# B&R Automation Studio project RTFProj (part 2)

#### calculation_displacementOfAxes.c
```c
/*********************************************************************************************
* B&R Automation - Perfection in Automation (https://www.br-automation.com)
    ******************************************************************************************
    * Program 	    : Master's Thesis - Soccer Table (Simulation)
    * Author  	    : Roman Parak
    * Created 	    : date ...
	* University    : Brno University of Technology(BUT)
	* Faculty       : Faculty of Mechanical Engineering(FME)
	* Study Program : Applied Computer Science and Control
	* Institute     : Institute of Automation and Computer Science
**********************************************************************************************
* Implementation OF PROGRAM simulation(rp_library/rp_funcx1/rp_functions.c)
**********************************************************************************************/

/************************************* LIBRARIES *********************************************/
#include <bur/plctypes.h>
#include <math.h>
#include <string.h>

#ifdef __cplusplus
	extern "C"
	{
#endif
	#include "rp_funcx1.h"
#ifdef __cplusplus
	};
#endif

void calculation_displacementOfAxes(struct calculation_displacementOfAxes* c_dOA)
{
	REAL max_dispOfD[4], min_dispOfD[4], max_posOfD[4], min_posOfD[4], matrix_posOfCPU[4][5], real_disp[4];
	REAL velocity[4], acceleration[4], deceleration[4];
	REAL aux_velocity[4], aux_acceleration[4];
	REAL aux_time;
	UDINT auxiliary_str;
	USINT i_rC, i_rCn, i, j, i_out, i_chRD, i_chRDn, i_chRDnn;

	struct calculation_realCrossing calc_rC;
	struct choosing_rightDummy ch_rightD;

	// Ceilings of the axes
	// Axes
	max_posOfD[0] = 820;
	max_posOfD[1] = 3050;
	max_posOfD[2] = 3050;
	max_posOfD[3] = 3055;

	min_posOfD[0] = -950;
	min_posOfD[1] = -3050;
	min_posOfD[2] = -3050;
	min_posOfD[3] = -3055;
	// Dummies
	max_dispOfD[0] = 820;
	max_dispOfD[1] = 1850;
	max_dispOfD[2] = 650;
	max_dispOfD[3] = 955;

	min_dispOfD[0] = -950;
	min_dispOfD[1] = -1850;
	min_dispOfD[2] = -650;
	min_dispOfD[3] = -955;
	// Actual positions of dummies CPU
	// goalkeeper
	matrix_posOfCPU[0][0] = 0 + c_dOA->act_displacementCPU[0];
	// defender
	matrix_posOfCPU[1][0] = -1200 + c_dOA->act_displacementCPU[1];
	matrix_posOfCPU[1][1] = 1200 + c_dOA->act_displacementCPU[1];
	// midfielder
	matrix_posOfCPU[2][0] = -2400 + c_dOA->act_displacementCPU[2];
	matrix_posOfCPU[2][1] = -1200 + c_dOA->act_displacementCPU[2];
	matrix_posOfCPU[2][2] = 0 + c_dOA->act_displacementCPU[2];
	matrix_posOfCPU[2][3] = 1200 + c_dOA->act_displacementCPU[2];
	matrix_posOfCPU[2][4] = 2400 + c_dOA->act_displacementCPU[2];
	// forward
	matrix_posOfCPU[3][0] = -2100 + c_dOA->act_displacementCPU[3];
	matrix_posOfCPU[3][1] = 0 + c_dOA->act_displacementCPU[3];
	matrix_posOfCPU[3][2] = 2100 + c_dOA->act_displacementCPU[3];

	// function block -> output is a array of real crossing
	calc_rC.tilted = c_dOA->tilted;
	auxiliary_str = (UDINT) strcpy(calc_rC.specific_direction,c_dOA->specific_direction);
	for(i_rC = 0; i_rC < (int)(sizeof(max_posOfD)/sizeof(max_posOfD[0])); i_rC++){
		calc_rC.act_posOfAxesCPU_Y[i_rC]		 = c_dOA->act_posOfAxesCPU_Y[i_rC];
		calc_rC.act_posOfAxesHUM_Y[i_rC]		 = c_dOA->act_posOfAxesHUM_Y[i_rC];
		calc_rC.count_axesIntersectionHUM[i_rC]  = c_dOA->count_axesIntersectionHUM[i_rC];
		calc_rC.reversed_HUM[i_rC]				 = c_dOA->reversed_HUM[i_rC];
	}
	for(i_rCn = 0; i_rCn < (int)(sizeof(c_dOA->act_posOfDummiesH)/sizeof(c_dOA->act_posOfDummiesH[0])); i_rCn++){
		calc_rC.act_posOfDummiesH[i_rCn] = c_dOA->act_posOfDummiesH[i_rCn];
	}
	calc_rC.x_posOfBall[0] = c_dOA->x_posOfBall[0];
	calc_rC.x_posOfBall[1] = c_dOA->x_posOfBall[1];
	calculation_realCrossing(&calc_rC);

	for(i = 0; i < (int)(sizeof(calc_rC.real_cross)/sizeof(calc_rC.real_cross[0])); i++){
		if(calc_rC.real_cross[i] > max_posOfD[i]){
			real_disp[i] = max_dispOfD[i];
		}else if(calc_rC.real_cross[i] < min_posOfD[i]){
			real_disp[i] = min_dispOfD[i];
		}else {
			ch_rightD.index      = i;
			ch_rightD.real_cross = calc_rC.real_cross[i];

			for(i_chRD = 0; i_chRD < (int)(sizeof(max_dispOfD)/sizeof(max_dispOfD[0])); i_chRD++){
				ch_rightD.max_dispOfD[i_chRD] = max_dispOfD[i_chRD];
				ch_rightD.min_dispOfD[i_chRD] = min_dispOfD[i_chRD];
			}

			for(i_chRDn = 0; i_chRDn < (int)(sizeof(max_dispOfD)/sizeof(max_dispOfD[0])); i_chRDn++){
				for(i_chRDnn = 0; i_chRDnn <= (int)(sizeof(max_dispOfD)/sizeof(max_dispOfD[0]));i_chRDnn++){
					ch_rightD.matrix_posOfCPU[i_chRDn][i_chRDnn] = matrix_posOfCPU[i_chRDn][i_chRDnn];
				}
			}
			choosing_rightDummy(&ch_rightD);

			real_disp[i] = ch_rightD.actual_displacement;
		}
	}// end for{i}

	for(i_out = 0; i_out < (int)(sizeof(calc_rC.real_cross)/sizeof(calc_rC.real_cross[0])); i_out++){
		// max velocity = 29000, max acceleration = 489 000
		aux_time = 0.07;
		aux_velocity[i_out] = fabs(fabs(real_disp[i_out]) - fabs(c_dOA->act_displacementCPU[i_out]))/c_dOA->time_axisIntersection[i_out];

		if(aux_velocity[i_out] > 29000){
			velocity[i_out] 		= fabs(fabs(real_disp[i_out]) - fabs(c_dOA->act_displacementCPU[i_out]))/aux_time;
			aux_acceleration[i_out] = velocity[i_out]/c_dOA->time_axisIntersection[i_out];

			if(aux_acceleration[i_out] > 489000){
				acceleration[i_out] = 489000;
				deceleration[i_out] = 489000;
			}else{
				acceleration[i_out] = aux_acceleration[i_out];
				deceleration[i_out] = aux_acceleration[i_out];
			}
		}else{
			velocity[i_out] 		= aux_velocity[i_out];
			aux_acceleration[i_out] = velocity[i_out]/c_dOA->time_axisIntersection[i_out];

			if(aux_acceleration[i_out] > 489000){
				acceleration[i_out] = 489000;
				deceleration[i_out] = 489000;
			}else{
				acceleration[i_out] = aux_acceleration[i_out];
				deceleration[i_out] = aux_acceleration[i_out];
			}
		}

		c_dOA->displacement[i_out] = real_disp[i_out];
		c_dOA->velocity[i_out] 	   = velocity[i_out];
		c_dOA->acceleration[i_out] = acceleration[i_out];
		c_dOA->deceleration[i_out] = deceleration[i_out];
	}// end for{i_out}

}// end function

void calculation_realCrossing(struct calculation_realCrossing* c_rC)
{
	REAL matrix_posOfHUM[4][5], matrix_crossH_Iter[0][5], matrix_crossH_Pos[0][5];
	REAL predicted_pos;
	USINT number_ofD[4], count_crossH, count_calcH;
	USINT iteration, iteration_positionH;
	USINT j, j_null, i_yC, i_yCn, i_cNC, i_out, r;
	BOOL auxiliary_bool,auxiliary_boolNo2;
	UDINT auxiliary_str;

	struct calculation_newCrossing calc_newC;

	auxiliary_bool 	  = 0;
	auxiliary_boolNo2 = 0;
	// Actual positions of dummies HUMAN
	// goalkeeper
	matrix_posOfHUM[0][0] = c_rC->act_posOfDummiesH[0];
	// defender
	matrix_posOfHUM[1][0] = c_rC->act_posOfDummiesH[1];
	matrix_posOfHUM[1][1] = c_rC->act_posOfDummiesH[2];
	// midfielder
	matrix_posOfHUM[2][0] = c_rC->act_posOfDummiesH[3];
	matrix_posOfHUM[2][1] = c_rC->act_posOfDummiesH[4];
	matrix_posOfHUM[2][2] = c_rC->act_posOfDummiesH[5];
	matrix_posOfHUM[2][3] = c_rC->act_posOfDummiesH[6];
	matrix_posOfHUM[2][4] = c_rC->act_posOfDummiesH[7];
	// forward
	matrix_posOfHUM[3][0] = c_rC->act_posOfDummiesH[8];
	matrix_posOfHUM[3][1] = c_rC->act_posOfDummiesH[9];
	matrix_posOfHUM[3][2] = c_rC->act_posOfDummiesH[10];

	number_ofD[0] = 1;
	number_ofD[1] = 2;
	number_ofD[2] = 5;
	number_ofD[3] = 3;

	calc_newC.reversed_HUM = 1;

	count_crossH   = c_rC->count_axesIntersectionHUM[0];
	count_calcH    = 5 - count_crossH;

	if(count_calcH == 0){
		iteration = 1;
	}else{
		iteration = count_calcH;
	}

	if(count_calcH < 5){
		for(j = 0; j < number_ofD[count_calcH - 1]; j++){
			if(c_rC->reversed_HUM[count_calcH - 1] == 0){
				if(((matrix_posOfHUM[count_calcH - 1][j] <= c_rC->act_posOfAxesHUM_Y[count_calcH - 1] + 100) && (matrix_posOfHUM[count_calcH - 1][j] >= c_rC->act_posOfAxesHUM_Y[count_calcH - 1])) && (matrix_posOfHUM[count_calcH - 1][j] != c_rC->act_posOfAxesHUM_Y[count_calcH - 1])){
					matrix_crossH_Iter[0][j] = count_calcH;
					matrix_crossH_Pos[0][j]  = fabs(fabs(matrix_posOfHUM[count_calcH - 1][j]) - fabs(c_rC->act_posOfAxesHUM_Y[count_calcH - 1]));
				}else if(((matrix_posOfHUM[count_calcH - 1][j] >= c_rC->act_posOfAxesHUM_Y[count_calcH - 1] - 100) && (matrix_posOfHUM[count_calcH - 1][j] <= c_rC->act_posOfAxesHUM_Y[count_calcH - 1])) && (matrix_posOfHUM[count_calcH - 1][j] != c_rC->act_posOfAxesHUM_Y[count_calcH - 1])){
					matrix_crossH_Iter[0][j] = count_calcH;
					matrix_crossH_Pos[0][j]  = (-1)*fabs(fabs(matrix_posOfHUM[count_calcH - 1][j]) - fabs(c_rC->act_posOfAxesHUM_Y[count_calcH - 1]));
				}else if(matrix_posOfHUM[count_calcH - 1][j] == c_rC->act_posOfAxesHUM_Y[count_calcH - 1]){
					matrix_crossH_Iter[0][j] = count_calcH;
					matrix_crossH_Pos[0][j]  = 0;
				}else{
					matrix_crossH_Iter[0][j] = 0;
					matrix_crossH_Pos[0][j]  = 0;
				}
			}else{
				matrix_crossH_Iter[0][j] = 0;
				matrix_crossH_Pos[0][j]  = 0;
			}
		}

		for(r = 0; r < number_ofD[count_calcH - 1]; r++){
			if(matrix_crossH_Iter[0][r] != 0){
				calc_newC.reversed_HUM = 0;
			}
		}
		for(j_null = 0; j_null < number_ofD[count_calcH - 1]; j_null++){
			if(matrix_crossH_Iter[0][j_null] != 0){
				auxiliary_bool 		= 1;
				predicted_pos  		= matrix_crossH_Pos[0][j_null];
				iteration_positionH = matrix_crossH_Iter[0][j_null];
			}
		}

		if(auxiliary_bool == 0){
			if(c_rC->tilted == 0){
				predicted_pos 		= 0;
				iteration_positionH = iteration;
			}else{
				auxiliary_boolNo2 = 1;
				for(i_yCn = 0; i_yCn < (int)(sizeof(c_rC->act_posOfAxesCPU_Y)/sizeof(c_rC->act_posOfAxesCPU_Y[0])); i_yCn++){
					c_rC->real_cross[i_yCn] = c_rC->act_posOfAxesCPU_Y[i_yCn];
				}
			}
		}

	}else{
		if(c_rC->tilted == 0){
			calc_newC.reversed_HUM = 0;
			predicted_pos 		   = 0;
			iteration_positionH    = count_calcH;
		}else{
			auxiliary_boolNo2 = 1;
			for(i_yC = 0; i_yC < (int)(sizeof(c_rC->act_posOfAxesCPU_Y)/sizeof(c_rC->act_posOfAxesCPU_Y[0])); i_yC++){
				c_rC->real_cross[i_yC] = c_rC->act_posOfAxesCPU_Y[i_yC];
			}
		}
	}// end : if(count_calcH < 5)

	if(auxiliary_boolNo2 != 1){
		auxiliary_str = (UDINT) strcpy(calc_newC.specific_direction,c_rC->specific_direction);
		calc_newC.iteration 		 = iteration_positionH;
		calc_newC.predicted_position = predicted_pos;
		for(i_cNC = 0; i_cNC < (int)(sizeof(c_rC->act_posOfAxesCPU_Y)/sizeof(c_rC->act_posOfAxesCPU_Y[0])); i_cNC++){
			calc_newC.act_posOfAxesCPU_Y[i_cNC] = c_rC->act_posOfAxesCPU_Y[i_cNC];
			calc_newC.act_posOfAxesHUM_Y[i_cNC] = c_rC->act_posOfAxesHUM_Y[i_cNC];
		}
		calc_newC.x_posOfBall[0] = c_rC->x_posOfBall[0];
		calc_newC.x_posOfBall[1] = c_rC->x_posOfBall[1];
		calculation_newCrossing(&calc_newC);

		for(i_out = 0; i_out < (int)(sizeof(c_rC->act_posOfAxesCPU_Y)/sizeof(c_rC->act_posOfAxesCPU_Y[0])); i_out++){
			c_rC->real_cross[i_out] = calc_newC.new_cross[i_out];
		}
	}// end if(auxiliary_boolNo2 != 1)
}// end function

void calculation_newCrossing(struct calculation_newCrossing* c_nC)
{
	INT gk_max, gk_min, value;
	SINT iteration;
	DINT resultUP, resultLF, resultDOWN, resultRH;
	REAL y_crossGK, y_crossDF, y_crossMD, y_crossFW;

	// initial max goalkeeper
	gk_max = 820;
	gk_min = -950;

	resultUP   = strcmp(c_nC->specific_direction, "up_backward");
	resultLF   = strcmp(c_nC->specific_direction, "left");
	resultDOWN = strcmp(c_nC->specific_direction, "down_backward");
	resultRH   = strcmp(c_nC->specific_direction, "right");

	if(resultUP == 0 || resultLF == 0){
		value = 200;
	}else if(resultDOWN == 0 || resultRH == 0){
		value = -200;
	}else{
		value = 200;
	}

	if(c_nC->iteration > 4){
		iteration = 4;
	}else{
		iteration = c_nC->iteration;
	}

	switch(iteration){
		case 1:
			{
				y_crossFW = c_nC->act_posOfAxesCPU_Y[4];
				y_crossMD = y_crossFW + value;
				y_crossDF = y_crossMD + value;
				y_crossGK = y_crossDF + value;

				if(fabs(y_crossGK) > fabs(y_crossFW)){
					y_crossGK = y_crossFW - value;
				}

				if(fabs(y_crossMD) < fabs(y_crossFW)){
					y_crossMD = y_crossFW - value;
					y_crossDF = y_crossMD - value;
				}
			}
			break;
		case 2:
			{
				if(c_nC->x_posOfBall[0] >= 9800){
					y_crossFW = c_nC->act_posOfAxesHUM_Y[iteration] - c_nC->predicted_position;
					y_crossMD = y_crossFW + value;
					y_crossDF = y_crossMD + value;
					y_crossGK = y_crossDF + value;

					if(fabs(y_crossGK) > fabs(y_crossFW)){
						y_crossGK = y_crossFW - value;
					}

					if(fabs(y_crossMD) < fabs(y_crossFW)){
						y_crossMD = y_crossFW - value;
						y_crossDF = y_crossMD - value;
					}
				}else{
					y_crossFW = c_nC->act_posOfAxesHUM_Y[3] - c_nC->predicted_position;
					y_crossMD = y_crossFW + value;
					y_crossDF = y_crossMD + value;
					y_crossGK = y_crossDF + value;

					if(fabs(y_crossGK) > fabs(y_crossFW)){
						y_crossGK = y_crossFW - value;
					}

					if(fabs(y_crossMD) < fabs(y_crossFW)){
						y_crossMD = y_crossFW - value;
						y_crossDF = y_crossMD - value;
					}
				}
			}
			break;
		case 3:
			{
				if(c_nC->reversed_HUM == 1){
					y_crossFW = c_nC->act_posOfAxesHUM_Y[3] - c_nC->predicted_position;
					y_crossMD = y_crossFW + value;
				}else{
					y_crossFW = c_nC->act_posOfAxesHUM_Y[3] - c_nC->predicted_position;
					y_crossMD = y_crossFW + value;
				}

				y_crossDF = y_crossMD + value;
				y_crossGK = y_crossFW + value;

				if(fabs(y_crossGK) > fabs(y_crossFW)){
					y_crossGK = y_crossFW - value;
				}

				if(fabs(y_crossMD) < fabs(y_crossFW)){
					y_crossMD = y_crossFW - value;
					y_crossDF = y_crossMD - value;
				}
			}
			break;
		case 4:
			{
				if(c_nC->x_posOfBall[0] >= 5300){
					if(c_nC->reversed_HUM == 1){
						y_crossFW = c_nC->act_posOfAxesCPU_Y[3] - c_nC->predicted_position;
						y_crossMD = c_nC->act_posOfAxesCPU_Y[2] - c_nC->predicted_position;
						y_crossDF = y_crossMD + value;
						y_crossGK = y_crossFW + value;
					}else{
						y_crossFW = c_nC->act_posOfAxesCPU_Y[3] - c_nC->predicted_position;
						y_crossMD = c_nC->act_posOfAxesCPU_Y[2] - c_nC->predicted_position;
						y_crossDF = y_crossMD - c_nC->predicted_position;
						y_crossGK = y_crossFW + value;

					}

					if(fabs(y_crossGK) > fabs(y_crossFW)){
						y_crossGK = y_crossFW - value;
					}
					if(fabs(y_crossMD) < fabs(y_crossFW)){
						y_crossDF = y_crossMD - value;
					}
				}else{
					y_crossFW = c_nC->act_posOfAxesCPU_Y[3] - c_nC->predicted_position;
					y_crossMD = c_nC->act_posOfAxesCPU_Y[2] - c_nC->predicted_position;
					y_crossDF = y_crossMD - c_nC->predicted_position;
					y_crossGK = y_crossFW + value;
				}

				if(c_nC->x_posOfBall[0] <= 2300){
					y_crossGK = c_nC->act_posOfAxesCPU_Y[0];
				}
			}
			break;
	}// end switch

	if(y_crossGK > gk_max){
		y_crossGK = y_crossDF - 200;
	}else if(y_crossGK < gk_min){
		y_crossGK = y_crossDF + 200;
	}

	c_nC->new_cross[0] = y_crossGK;
	c_nC->new_cross[1] = y_crossDF;
	c_nC->new_cross[2] = y_crossMD;
	c_nC->new_cross[3] = y_crossFW;

}// end function

void choosing_rightDummy(struct choosing_rightDummy* ch_rD)
{
	REAL real_cross;
	REAL d_DFD[2],d_MDD[5], d_FWD[3];
	USINT i_df, i_md, i_fw;
	struct calculete_min calc_m;

	switch(ch_rD->index){
		case 0:
			{
				real_cross 				   = ch_rD->real_cross;
				ch_rD->actual_displacement = real_cross;
			}
			break;
		case 1:
			{
				d_DFD[0] = fabs((fabs(ch_rD->matrix_posOfCPU[ch_rD->index][0]) + ch_rD->real_cross));
				d_DFD[1] = fabs((ch_rD->matrix_posOfCPU[ch_rD->index][1] - ch_rD->real_cross));

				for(i_df = 0; i_df < (int)(sizeof(calc_m.cmp_num)/sizeof(calc_m.cmp_num[0])); i_df++){
					if(i_df < ((int)(sizeof(d_DFD)/sizeof(d_DFD[0])))){
						calc_m.cmp_num[i_df] = d_DFD[i_df];
					}else{
						calc_m.cmp_num[i_df] = 5000;
					}
				}
			}
			break;
		case 2:
			{
				d_MDD[0] = fabs((fabs(ch_rD->matrix_posOfCPU[ch_rD->index][0]) + ch_rD->real_cross));
				d_MDD[1] = fabs((fabs(ch_rD->matrix_posOfCPU[ch_rD->index][1]) + ch_rD->real_cross));
				d_MDD[2] = fabs((ch_rD->real_cross));
				d_MDD[3] = fabs((fabs(ch_rD->matrix_posOfCPU[ch_rD->index][3]) - ch_rD->real_cross));
				d_MDD[4] = fabs((fabs(ch_rD->matrix_posOfCPU[ch_rD->index][4]) - ch_rD->real_cross));

				for(i_md = 0; i_md < (int)(sizeof(calc_m.cmp_num)/sizeof(calc_m.cmp_num[0])); i_md++){
					calc_m.cmp_num[i_md] = d_MDD[i_md];
				}
			}
			break;
		case 3:
			{
				d_FWD[0] = fabs((fabs(ch_rD->matrix_posOfCPU[ch_rD->index][0]) + ch_rD->real_cross));
				d_FWD[1] = fabs((ch_rD->real_cross));
				d_FWD[2] = fabs((fabs(ch_rD->matrix_posOfCPU[ch_rD->index][2]) - ch_rD->real_cross));

				for(i_fw = 0; i_fw < (int)(sizeof(calc_m.cmp_num)/sizeof(calc_m.cmp_num[0])); i_fw++){
					if(i_fw < ((int)(sizeof(d_FWD)/sizeof(d_FWD[0])))){
						calc_m.cmp_num[i_fw] = d_FWD[i_fw];
					}else{
						calc_m.cmp_num[i_fw] = 5000;
					}
				}
			}
			break;
	}// end switch

	if(ch_rD->index != 0){
		calculete_min(&calc_m);

		if(calc_m.number > ch_rD->max_dispOfD[ch_rD->index]){
			real_cross = ch_rD->max_dispOfD[ch_rD->index];
		}else if(calc_m.number < ch_rD->min_dispOfD[ch_rD->index]){
			real_cross = ch_rD->min_dispOfD[ch_rD->index];
		}else{
			real_cross = calc_m.number;
		}

		if(ch_rD->real_cross > ch_rD->matrix_posOfCPU[ch_rD->index][calc_m.index]){
			ch_rD->actual_displacement = real_cross;
		}else{
			ch_rD->actual_displacement = (-1)*real_cross;
		}
	}
}// end function

void calculete_min(struct calculete_min* c_m)
{
	REAL min;
	USINT i, idx;

	min = 30000;
	for(i = 0; i < (int)(sizeof(c_m->cmp_num)/sizeof(c_m->cmp_num[0])); i++){
		if(c_m->cmp_num[i] < min){
			min = c_m->cmp_num[i];
			idx = i;
		}
	}

	c_m->index  = idx;
	c_m->number = min;
}// end function
```

#### measurement_ofScore.c
```c
#include <bur/plctypes.h>
#include <bur/plc.h>
#include <astime.h>
#include <string.h>
#include <math.h>

#ifdef __cplusplus
	extern "C"
	{
#endif
	#include "rp_funcx1.h"
#ifdef __cplusplus
	};
#endif
void initialization(struct measurement_ofScore* m_oS);

void measurement_ofScore(struct measurement_ofScore* m_oS)
{

    if(!m_oS->start_measurement){
        initialization(m_oS);
    }

    switch(m_oS->Internal.state){
        case 0:
            {
                if(m_oS->Internal.counter <= 0){
                    m_oS->Internal.counter = 0;
                }

                m_oS->Internal.results[0]   = strcmp(m_oS->PLAYER1_NAME, "");
                m_oS->Internal.results[1]   = strcmp(m_oS->PLAYER2_NAME, "");

                if(m_oS->start_measurement == 1 && m_oS->Error == 0){
                    if(m_oS->Internal.results[0] == 0 && m_oS->Internal.results[1] == 0){
                        m_oS->Internal.auxiliary_str[5] = (UDINT) strcpy(m_oS->PLAYER1_NAME,"PLAYER 1");
                        m_oS->Internal.auxiliary_str[6] = (UDINT) strcpy(m_oS->PLAYER2_NAME,"PLAYER 2");
                    }
                    // CPU NAME
                    m_oS->Internal.auxiliary_str[7] = (UDINT) strcpy(m_oS->team_nameCPU,"B&R ROBOT");
                    // HUMAN NAME
                    strcpy(m_oS->Internal.string[5],m_oS->PLAYER1_NAME);
                    strcpy(m_oS->Internal.string[6]," \n \t& \n");
                    strcpy(m_oS->Internal.string[8], m_oS->PLAYER2_NAME);
                    m_oS->Internal.auxiliary_str[8] = (UDINT) strcat(m_oS->Internal.string[5], m_oS->Internal.string[6]);
                    strcpy(m_oS->Internal.string[7], m_oS->Internal.string[5]);
                    m_oS->Internal.auxiliary_str[9] = (UDINT) strcat(m_oS->Internal.string[7], m_oS->Internal.string[8]);
                    m_oS->Internal.auxiliary_str[10] = (UDINT) strcpy(m_oS->team_nameHUM,m_oS->Internal.auxiliary_str[9]);
                    // CHANGE STATE
                    m_oS->Internal.state = 1;
                }else if(m_oS->Error == 1){
                    m_oS->Internal.state = 5;
                }else if(m_oS->pause == 1){
                    m_oS->Internal.before_state = m_oS->Internal.state;
                    m_oS->Internal.state = 6;
                }else{
                    m_oS->Internal.state = 0;
                }
            }
            break;
        case 1:
            {
                if(m_oS->sens_wicket_CPU == 1){
                    m_oS->count_goals_CPU++;
                    m_oS->sens_wicket_CPU = 0;
                }

                if(m_oS->sens_wicket_HUM == 1){
                    m_oS->count_goals_HUM++;
                    m_oS->sens_wicket_HUM = 0;
                }

                if((m_oS->count_goals_HUM - m_oS->count_goals_CPU) == 0){
                    m_oS->probability_CPU = 50;
                    m_oS->probability_HUM = 50;
                }else if((m_oS->count_goals_HUM - m_oS->count_goals_CPU) < 0){
                    if(fabs((m_oS->count_goals_HUM - m_oS->count_goals_CPU)) <= 5){
                        m_oS->probability_CPU = 50 + fabs((m_oS->count_goals_HUM - m_oS->count_goals_CPU))*10;
                        m_oS->probability_HUM = 100 - m_oS->probability_CPU;
                    }else{
                        m_oS->probability_CPU = 100;
                        m_oS->probability_HUM = 0;
                    }
                }else{
                    if(fabs((m_oS->count_goals_HUM - m_oS->count_goals_CPU)) <= 5){
                        m_oS->probability_HUM = 50 + fabs((m_oS->count_goals_HUM - m_oS->count_goals_CPU))*10;
                        m_oS->probability_CPU = 100 - m_oS->probability_HUM;
                    }else{
                        m_oS->probability_HUM = 100;
                        m_oS->probability_CPU = 0;
                    }
                }
                if(((m_oS->count_goals_CPU + m_oS->count_goals_HUM) == 10) && m_oS->Error == 0){
                    m_oS->Internal.state             = 2;
                    m_oS->Internal.write_matchInfo   = 1;
                }else if(m_oS->exit_game == 1 ){
                    m_oS->Internal.state = 3;
                }else if(m_oS->restart_measurement == 1){
                    m_oS->Internal.state = 4;
                }else if(m_oS->Error == 1){
                    m_oS->Internal.state = 5;
                }else if(m_oS->pause == 1){
                    m_oS->Internal.before_state = m_oS->Internal.state;
                    m_oS->Internal.state = 6;
                }else{
                    m_oS->Internal.state = 1;
                }

            }
            break;
        case 2:
            {
                if(m_oS->Internal.write_matchInfo == 1){
                    // call FB : Get time and date
                    m_oS->Internal.UtcDTStructureGetTime_1.enable = 1;
                    m_oS->Internal.UtcDTStructureGetTime_1.pDTStructure = (UDINT) &m_oS->Internal.DTStruct;
                    UtcDTStructureGetTime(&m_oS->Internal.UtcDTStructureGetTime_1);
                    ascDTStructure((UDINT) &m_oS->Internal.DTStruct, (UDINT) &m_oS->Internal.string[0], m_oS->Internal.length);
                    // write time and date into the variable
                    m_oS->Internal.auxiliary_str[0] = (UDINT) strcpy(m_oS->match_informations.date[m_oS->Internal.counter],m_oS->Internal.string[0]);
                    // write score
                    m_oS->match_informations.score_CPU[m_oS->Internal.counter] = m_oS->count_goals_CPU;
                    m_oS->match_informations.score_HUM[m_oS->Internal.counter] = m_oS->count_goals_HUM;
                    // write name of B&R team
                    m_oS->Internal.auxiliary_str[1] = (UDINT) strcpy(m_oS->match_informations.team_name_CPU[m_oS->Internal.counter],"B&R ROBOT");
                    // write names of both players
                    strcpy(m_oS->Internal.string[1],m_oS->PLAYER1_NAME);
                    strcpy(m_oS->Internal.string[2]," & ");
                    strcpy(m_oS->Internal.string[4], m_oS->PLAYER2_NAME);
                    m_oS->Internal.auxiliary_str[2] = (UDINT) strcat(m_oS->Internal.string[1], m_oS->Internal.string[2]);
                    strcpy(m_oS->Internal.string[3], m_oS->Internal.string[1]);
                    m_oS->Internal.auxiliary_str[3] = (UDINT) strcat(m_oS->Internal.string[3], m_oS->Internal.string[4]);
                    m_oS->Internal.auxiliary_str[4] = (UDINT) strcpy(m_oS->match_informations.team_name_HUM[m_oS->Internal.counter],m_oS->Internal.auxiliary_str[3]);

                    m_oS->Internal.counter++;
                    m_oS->Internal.write_matchInfo = 0;
                }

                if(m_oS->exit_game == 1){
                    m_oS->Internal.state = 3;
                }else if(m_oS->restart_measurement == 1){
                    m_oS->Internal.state = 4;
                }else if(m_oS->Error == 1){
                    m_oS->Internal.state = 5;
                }else if(m_oS->pause == 1){
                    m_oS->Internal.before_state = m_oS->Internal.state;
                    m_oS->Internal.state = 6;
                }else{
                    m_oS->Internal.state = 2;
                }
            }
            break;
        case 3:
            {
                // exit game
                m_oS->start_measurement   = 0;
                m_oS->exit_game           = 0;
                m_oS->restart_measurement = 0;
                m_oS->count_goals_CPU     = 0;
                m_oS->count_goals_HUM     = 0;

                m_oS->Internal.e_r_str[0] = (UDINT) strcpy(m_oS->PLAYER1_NAME,"");
                m_oS->Internal.e_r_str[1] = (UDINT) strcpy(m_oS->PLAYER2_NAME,"");

                if(m_oS->Error == 1){
                    m_oS->Internal.state = 5;
                }else if(m_oS->pause == 1){
                    m_oS->Internal.before_state = m_oS->Internal.state;
                    m_oS->Internal.state = 6;
                }else{
                    m_oS->Internal.state = 0;
                }
            }
            break;
        case 4:
            {
                // restart game
                m_oS->start_measurement   = 0;
                m_oS->exit_game           = 0;
                m_oS->restart_measurement = 0;
                m_oS->count_goals_CPU     = 0;
                m_oS->count_goals_HUM     = 0;

                m_oS->Internal.e_r_str[2] = (UDINT) strcpy(m_oS->PLAYER1_NAME,m_oS->PLAYER1_NAME);
                m_oS->Internal.e_r_str[3] = (UDINT) strcpy(m_oS->PLAYER2_NAME,m_oS->PLAYER2_NAME);

                if(m_oS->Error == 1){
                    m_oS->Internal.state = 5;
                }else if(m_oS->pause == 1){
                    m_oS->Internal.before_state = m_oS->Internal.state;
                    m_oS->Internal.state = 6;
                }else{
                    m_oS->Internal.state = 1;
                }
            }
            break;
        case 5:
            {
                // error state
                if(m_oS->Error == 0){
                    m_oS->Internal.state = 3;
                }else if(m_oS->pause == 1){
                    m_oS->Internal.before_state = m_oS->Internal.state;
                    m_oS->Internal.state = 6;
                }
            }
            break;
        case 6:
            {
                // pause
                if(m_oS->Error == 1){
                    m_oS->Internal.state = 5;
                }else if(m_oS->pause == 0){
                    m_oS->Internal.state = m_oS->Internal.before_state;
                }
            }
            break;
    }// end switch

}// end fucntion

void initialization(struct measurement_ofScore* m_oS){
    m_oS->Internal.state             = 0;
    m_oS->Internal.e_r_str[0]        = 0;
    m_oS->Internal.e_r_str[1]        = 0;
    m_oS->Internal.e_r_str[2]        = 0;
    m_oS->Internal.e_r_str[3]        = 0;
    m_oS->Internal.auxiliary_str[0]  = 0;
    m_oS->Internal.auxiliary_str[1]  = 0;
    m_oS->Internal.auxiliary_str[2]  = 0;
    m_oS->Internal.auxiliary_str[3]  = 0;
    m_oS->Internal.auxiliary_str[4]  = 0;
    m_oS->Internal.auxiliary_str[5]  = 0;
    m_oS->Internal.auxiliary_str[6]  = 0;
    m_oS->Internal.auxiliary_str[7]  = 0;
    m_oS->Internal.auxiliary_str[8]  = 0;
    m_oS->Internal.auxiliary_str[9]  = 0;
    m_oS->Internal.auxiliary_str[10] = 0;
    m_oS->Internal.counter           = 0;
    m_oS->Internal.length            = 25;
    m_oS->Internal.write_matchInfo   = 0;
    m_oS->Internal.results[0]        = 0;
    m_oS->Internal.results[1]        = 0;
	m_oS->Internal.before_state      = 0;
    m_oS->count_goals_CPU            = 0;
    m_oS->count_goals_HUM            = 0;
    m_oS->sens_wicket_HUM            = 0;
    m_oS->restart_measurement        = 0;
    m_oS->pause                      = 0;
    m_oS->exit_game                  = 0;
    m_oS->start_measurement          = 0;
    m_oS->probability_CPU            = 50;
    m_oS->probability_HUM            = 50;
}// end function
```

#### start_linearAxis.c
```c
#include <bur/plctypes.h>
#include <stdio.h>
#include <stdlib.h>
#include <MpAxis.h>

#ifdef __cplusplus
	extern "C"
	{
#endif
	#include "rp_funcx1.h"
#ifdef __cplusplus
	};
#endif
void initialization_sla(struct start_linearAxis* s_la);

void start_linearAxis(struct start_linearAxis* s_la)
{
	if(!s_la->Enable){
		initialization_sla(s_la);
	}

	switch(s_la->Internal.state){
		case 0:
			{
				s_la->Internal.before_state     = s_la->Internal.state;

				if(s_la->start_btn == 1){
					// adjustment parameters -> axis
					s_la->axis_param->Home.Mode 				  = mpAXIS_HOME_MODE_BLOCK_TORQUE;
					s_la->axis_param->Home.Position 		  	  = s_la->max_leftPosition;
					s_la->axis_param->Home.StartVelocity   		  = s_la->velocity;
					s_la->axis_param->Home.HomingVelocity  		  = s_la->velocity;
					s_la->axis_param->Home.Acceleration    		  = 200000;
					s_la->axis_param->Home.StartDirection  		  = mpAXIS_HOME_DIR_POSITIVE;
					s_la->axis_param->Home.HomingDirection 		  = mpAXIS_HOME_DIR_NEGATIVE;
					s_la->axis_param->Home.TorqueLimit	 		  = 0.02;
					s_la->axis_param->Home.PositionErrorStopLimit = s_la->max_leftPosition + 10;
					// reset output
					s_la->succesfully = 0;
					if(s_la->axis_name->Error == 1 || s_la->axis_name->StatusID != 0){
						s_la->axis_name->ErrorReset = 0;
						if(s_la->axis_name->ErrorReset == 0){
							s_la->Internal.state = 10;
						}
					}else{
						if(s_la->start_btn == 1){
							s_la->Internal.state = 1;
						}
					}
				}
			}
			break;
		case 1:
			{
				s_la->Internal.before_state = s_la->Internal.state;
				// power on -> axis
				s_la->axis_name->Power = 1;

				if(s_la->axis_name->Error == 1 || s_la->axis_name->StatusID != 0){
					s_la->axis_name->ErrorReset = 0;
					if(s_la->axis_name->ErrorReset == 0){
						s_la->Internal.state = 10;
					}
				}else{
					if(s_la->axis_name->PowerOn == 1){
						s_la->Internal.state = 2;
					}
				}
			}
			break;
		case 2:
			{
				s_la->Internal.before_state = s_la->Internal.state;
				// update -> axis
				s_la->axis_name->Update = 1;

				if(s_la->axis_name->Error == 1 || s_la->axis_name->StatusID != 0){
					s_la->axis_name->ErrorReset = 0;
					if(s_la->axis_name->ErrorReset == 0){
						s_la->Internal.state = 10;
					}
				}else{
					if(s_la->axis_name->UpdateDone == 1){
						s_la->axis_name->Update = 0;
						if(s_la->axis_name->UpdateDone == 0){
							s_la->Internal.state 	= 3;
						}
					}
				}
			}
		case 3:
			{
				s_la->Internal.before_state = s_la->Internal.state;
				// home -> axis
				s_la->axis_name->Home = 1;

				if(s_la->axis_name->Error == 1 || s_la->axis_name->StatusID != 0){
					s_la->axis_name->ErrorReset = 0;
					if(s_la->axis_name->ErrorReset == 0){
						s_la->Internal.state = 10;
					}
				}else{
					if(s_la->axis_name->IsHomed == 1){
						s_la->axis_name->Home = 0;
						s_la->succesfully     = 1;
						s_la->Internal.state  = 0;
					}
				}
			}
			break;
		case 10:
			{
				s_la->axis_name->ErrorReset = 1;

				if(s_la->axis_name->Error == 1 || s_la->axis_name->StatusID != 0){
					s_la->Internal.state = 10;
				}else{
					s_la->axis_name->ErrorReset = 0;
					s_la->Internal.state 		= s_la->Internal.before_state;
				}
			}
			break;
	}// end switch
}// end function

void initialization_sla(struct start_linearAxis* s_la)
{
	s_la->Internal.state 		= 0;
	s_la->Internal.before_state = 0;
	s_la->start_btn				= 0;
	s_la->succesfully     		= 0;
}// end function
```

#### start_rotaryAxis.c
```c
#include <bur/plctypes.h>
#include <stdio.h>
#include <stdlib.h>
#include <MpAxis.h>

#ifdef __cplusplus
	extern "C"
	{
#endif
	#include "rp_funcx1.h"
#ifdef __cplusplus
	};
#endif
void initialization_sra(struct start_rotaryAxis* s_ra);

void start_rotaryAxis(struct start_rotaryAxis* s_ra)
{
	if(!s_ra->Enable){
		initialization_sra(s_ra);
	}

	switch(s_ra->Internal.state){
		case 0:
			{
				s_ra->Internal.before_state     = s_ra->Internal.state;

				if(s_ra->start_btn == 1){
					// adjust param -> axis
					// move position
					s_ra->axis_param->Acceleration = 3969754;
					s_ra->axis_param->Deceleration = 3969754;
					s_ra->axis_param->Velocity     = 1000;
					s_ra->axis_param->Position 	   = 0;
					// home
					s_ra->axis_param->Home.Position = s_ra->value_ofRotatation;
					// reset output
					s_ra->succesfully = 0;
					if(s_ra->axis_name->Error == 1 || s_ra->axis_name->StatusID != 0){
						s_ra->axis_name->ErrorReset = 0;
						if(s_ra->axis_name->ErrorReset == 0){
							s_ra->Internal.state = 10;
						}
					}else{
						if(s_ra->start_btn == 1){
							s_ra->Internal.state = 1;
						}
					}
				}
			}
			break;
		case 1:
			{
				s_ra->Internal.before_state = s_ra->Internal.state;
				// power on -> axis
				s_ra->axis_name->Power = 1;

				if(s_ra->axis_name->Error == 1 || s_ra->axis_name->StatusID != 0){
					s_ra->axis_name->ErrorReset = 0;
					if(s_ra->axis_name->ErrorReset == 0){
						s_ra->Internal.state = 10;
					}
				}else{
					if(s_ra->axis_name->PowerOn == 1){
						s_ra->Internal.state = 2;
					}
				}
			}
			break;
		case 2:
			{
				s_ra->Internal.before_state = s_ra->Internal.state;
				// update -> axis
				s_ra->axis_name->Update = 1;

				if(s_ra->axis_name->Error == 1 || s_ra->axis_name->StatusID != 0){
					s_ra->axis_name->ErrorReset = 0;
					if(s_ra->axis_name->ErrorReset == 0){
						s_ra->Internal.state = 10;
					}
				}else{
					if(s_ra->axis_name->UpdateDone == 1){
						s_ra->axis_name->Update = 0;
						if(s_ra->axis_name->Update == 0){
							s_ra->Internal.state = 3;
						}
					}
				}
			}
		case 3:
			{
				s_ra->Internal.before_state = s_ra->Internal.state;
				// home -> axis
				s_ra->axis_name->Home = 1;

				if(s_ra->axis_name->Error == 1 || s_ra->axis_name->StatusID != 0){
					s_ra->axis_name->ErrorReset = 0;
					if(s_ra->axis_name->ErrorReset == 0){
						s_ra->Internal.state = 10;
					}
				}else{
					if(s_ra->axis_name->IsHomed == 1){
						s_ra->axis_name->Home = 0;
						s_ra->Internal.state  = 4;
					}
				}
			}
			break;
		case 4:
			{
				s_ra->Internal.before_state = s_ra->Internal.state;
				// move absolute -> axis
				s_ra->axis_name->MoveAbsolute = 1;

				if(s_ra->axis_name->Error == 1 || s_ra->axis_name->StatusID != 0){
					s_ra->axis_name->ErrorReset = 0;
					if(s_ra->axis_name->ErrorReset == 0){
						s_ra->Internal.state = 10;
					}
				}else{
					if(s_ra->axis_name->InPosition == 1){
						s_ra->axis_name->MoveAbsolute = 0;

						if(s_ra->axis_name->MoveAbsolute == 0){
							s_ra->succesfully	 = 1;
							s_ra->Internal.state = 0;
						}
					}
				}
			}
			break;
		case 10:
			{
				s_ra->axis_name->ErrorReset = 1;

				if(s_ra->axis_name->Error == 1 || s_ra->axis_name->StatusID != 0){
					s_ra->Internal.state = 10;
				}else{
					s_ra->axis_name->ErrorReset = 0;
					s_ra->Internal.state 		= s_ra->Internal.before_state;
				}
			}
			break;
	}// end switch
}// end function

void initialization_sra(struct start_rotaryAxis* s_ra)
{
	s_ra->Internal.state 		= 0;
	s_ra->Internal.before_state = 0;
	s_ra->start_btn				= 0;
	s_ra->succesfully     		= 0;
}// end function
```

#### err_detection.c
```c
#include <bur/plctypes.h>
#ifdef __cplusplus
	extern "C"
	{
#endif
	#include "rp_funcx1.h"
#ifdef __cplusplus
	};
#endif

void err_detection(struct err_detection* e_d)
{
	USINT i, count_err;

	for(i = 0; i < (int)(sizeof(e_d->rotary_ERR)/sizeof(e_d->rotary_ERR[0])); i++){
		if((e_d->rotary_ERR[i] || e_d->linear_ERR[i]) == 1){
			count_err++;
		}
	}

	if(count_err != 0){
		e_d->err_detect = 1;
	}else{
		e_d->err_detect = 0;
	}
}
```

#### control_temperature.c
```c
#include <bur/plctypes.h>
#ifdef __cplusplus
	extern "C"
	{
#endif
	#include "rp_funcx1.h"
#ifdef __cplusplus
	};
#endif

void control_temperature(struct control_temperature* c_t)
{
	USINT i;
	USINT MAX_TEMPERATURE_ROTARY = 100, MAX_TEMPERATURE_LINEAR = 100;

	for(i = 0; i < (int)(sizeof(c_t->temperature_rotary)/sizeof(c_t->temperature_rotary[0])); i++){
		if(c_t->temperature_rotary[i] >= MAX_TEMPERATURE_ROTARY){
			c_t->high_temp_rotary[i] = 1;
		}else{
			c_t->high_temp_rotary[i] = 0;
		}

		if(c_t->temperature_linear[i] >= MAX_TEMPERATURE_LINEAR){
			c_t->high_temp_linear[i] 	 = 1;
			c_t->start_cooling_linear[i] = 1;
		}else{
			c_t->high_temp_linear[i] 	 = 0;
			c_t->start_cooling_linear[i] = 0;
		}
	}
}
```

#### ball_shooting.c
```c
#include <bur/plctypes.h>
#include <stdio.h>
#include <stdlib.h>
#include <MpAxis.h>

#ifdef __cplusplus
	extern "C"
	{
#endif
	#include "rp_funcx1.h"
#ifdef __cplusplus
	};
#endif
void init_ball_shooting(struct ball_shooting* b_s);
void ball_shooting(struct ball_shooting* b_s)
{
	if(b_s->Enable == 0){
		init_ball_shooting(&b_s);
	}

	switch(b_s->Internal.state){
		case 0:
			{
				if(b_s->start_shoot == 1){
					// initialization parameters of axes for shooting ball
					b_s->rotary_axes->CyclicPosition = 1;
					b_s->rotary_axes->Position		 = -500;
					b_s->rotary_axes->Velocity 		 = 63000;

					// change state
					b_s->Internal.state = 1;
				}
			}
			break;
		case 1:
			{
				if(b_s->rotary_axes->Info.SlavePosition == b_s->rotary_axes->Position){
					// second position
					b_s->rotary_axes->Position	= 500;
					if(b_s->rotary_axes->Info.SlavePosition == 500){
						b_s->Internal.state = 2;
					}
				}
			}
			break;
		case 2:
			{
				if(b_s->rotary_axes->Info.SlavePosition == b_s->rotary_axes->Position){
					// second position
					b_s->rotary_axes->Position	= -250;

					if(b_s->rotary_axes->Info.SlavePosition == -250){
						b_s->successfully = 1;
						if(b_s->successfully == 1){
							b_s->Internal.state = 0;
						}
					}
				}

			}
			break;
	}// end switch
}// end function

void init_ball_shooting(struct ball_shooting* b_s)
{
	b_s->Internal.state = 0;
	b_s->successfully   = 0;
	b_s->start_shoot    = 0;
}
```

#### turn_position.c
```c
#include <bur/plctypes.h>
#include <stdio.h>
#include <stdlib.h>
#include <MpAxis.h>

#ifdef __cplusplus
	extern "C"
	{
#endif
	#include "rp_funcx1.h"
#ifdef __cplusplus
	};
#endif
void initial_turn_pos(struct turn_position* t_p);
void turn_position(struct turn_position* t_p)
{
	if(t_p->Enable == 0){
		initial_turn_pos(&t_p);
	}

	switch(t_p->Internal.state){
		case 0:
			{
				// parameters of move
				t_p->Internal.distance_ofMovePos  = 100 + 170 + 80 + 150;
				t_p->Internal.distance_ofMoveNeg  = (-1)*t_p->Internal.distance_ofMovePos;
				// velocity
				t_p->rotary_axes->Velocity 		= 1500;
				t_p->linear_axes->Velocity 		= 500;
				// initialization parameters
				t_p->Internal.max_pos_ofAxes[0] = 800;
				t_p->Internal.max_pos_ofAxes[1] = 1030;
				t_p->Internal.max_pos_ofAxes[2] = 520;
				t_p->Internal.max_pos_ofAxes[3] = 830;

				t_p->Internal.min_pos_ofAxes[0] = -910;
				t_p->Internal.min_pos_ofAxes[1] = -930;
				t_p->Internal.min_pos_ofAxes[2] = -500;
				t_p->Internal.min_pos_ofAxes[3] = -770;

				// start function
				if(t_p->start_turn == 1){
					t_p->successfully = 0;
					if(t_p->successfully == 0){
						// first position
						t_p->rotary_axes->Position = 500;
						if((t_p->linear_axes->Info.SlavePosition + t_p->Internal.distance_ofMovePos) > t_p->Internal.max_pos_ofAxes[t_p->index_ofAxis]){
							t_p->Internal.auxiliary_move_pos = t_p->linear_axes->Info.SlavePosition;
							t_p->linear_axes->Position = t_p->linear_axes->Info.SlavePosition + t_p->Internal.distance_ofMoveNeg;
						}else if((t_p->linear_axes->Info.SlavePosition + t_p->Internal.distance_ofMovePos) < t_p->Internal.min_pos_ofAxes[t_p->index_ofAxis]){
							t_p->Internal.auxiliary_move_pos = t_p->linear_axes->Info.SlavePosition;
							t_p->linear_axes->Position = t_p->linear_axes->Info.SlavePosition + t_p->Internal.distance_ofMovePos;
						}else{
							t_p->Internal.auxiliary_move_pos = t_p->linear_axes->Info.SlavePosition;
							t_p->linear_axes->Position = t_p->linear_axes->Info.SlavePosition + t_p->Internal.distance_ofMovePos;
						}
						// change state
						t_p->Internal.state = 1;

					}
				}
			}
			break;
		case 1:
			{

				if((t_p->rotary_axes->Position == t_p->rotary_axes->Info.SlavePosition) &&(t_p->linear_axes->Position == t_p->linear_axes->Info.SlavePosition)){
					t_p->rotary_axes->Position = -500;
					t_p->Internal.state = 2;
				}

			}
			break;
		case 2:
			{
				if((t_p->rotary_axes->Position == t_p->rotary_axes->Info.SlavePosition) &&(t_p->linear_axes->Position == t_p->linear_axes->Info.SlavePosition)){
					// initial position
					t_p->linear_axes->Position = t_p->Internal.distance_ofMoveNeg;
					t_p->rotary_axes->Position = -250;
					// change state
					t_p->Internal.state = 3;
				}

			}
			break;
		case 3:
			{
				if((t_p->rotary_axes->Position == t_p->rotary_axes->Info.SlavePosition) &&(t_p->linear_axes->Position == t_p->linear_axes->Info.SlavePosition)){
					t_p->successfully = 1;
					t_p->Internal.state = 0;
				}

			}
			break;
	}// end switch
}// end function

void initial_turn_pos(struct turn_position* t_p)
{
	t_p->Internal.state = 0;
	t_p->successfully   = 0;
	t_p->start_turn		= 0;
}
```

#### check_attack_mode.c
```c
#include <bur/plctypes.h>
#ifdef __cplusplus
	extern "C"
	{
#endif
	#include "rp_funcx1.h"
#ifdef __cplusplus
	};
#endif

void check_attack_mode(struct check_attack_mode* ch_aM)
{
	struct calculation_posDummies calculation_posDummies_0;
	struct detect_axisNumber detect_axisNumber_0;
	struct choose_attack_mode choose_attack_mode_0;
	INT behind_position, before_position;
	USINT i_chp, i_aM, stand_mode;
	REAL max_pos[4], min_pos[4];

	max_pos[0] = 800;
	max_pos[1] = 1060;
	max_pos[2] = 550;
	max_pos[3] = 860;

	min_pos[0] = -910;
	min_pos[1] = -960;
	min_pos[2] = -530;
	min_pos[3] = -800;

	for(i_chp = 0; i_chp < (int)(sizeof(ch_aM->act_displacement_cpu)/sizeof(ch_aM->act_displacement_cpu[0])); i_chp++){
		calculation_posDummies_0.displacement[i_chp] = ch_aM->act_displacement_cpu[i_chp];
		calculation_posDummies_0.max_disp[i_chp]	 = max_pos[i_chp];
		calculation_posDummies_0.min_disp[i_chp]	 = min_pos[i_chp];
	}

	calculation_posDummies(&calculation_posDummies_0);

	detect_axisNumber_0.ball1_x = ch_aM->ball1_x;
	detect_axisNumber_0.ball2_x = ch_aM->ball2_x;
	detect_axisNumber(&detect_axisNumber_0);

	if(detect_axisNumber_0.axis_number != 10){
		if(ch_aM->angle_ofRotation[detect_axisNumber_0.axis_number] > 0){
			// stand before the ball
			behind_position = -90;
			before_position = 90;
			stand_mode		= 1;
		}else{
			// stand behind the ball
			behind_position = -200; // -170
			before_position = 350;  // 320
			stand_mode		= 2;
		}

		for(i_aM = 0; i_aM < (int)(sizeof(calculation_posDummies_0.actual_positionsOfDummies)/sizeof(calculation_posDummies_0.actual_positionsOfDummies[0])); i_aM++){
			choose_attack_mode_0.actual_positionsOfDummies[i_aM] = calculation_posDummies_0.actual_positionsOfDummies[i_aM];
		}
		choose_attack_mode_0.ball1_x 		 = ch_aM->ball1_x;
		choose_attack_mode_0.ball1_y 		 = ch_aM->ball1_y;
		choose_attack_mode_0.ball2_x 		 = ch_aM->ball2_x;
		choose_attack_mode_0.ball2_y 		 = ch_aM->ball2_y;
		choose_attack_mode_0.axis_number 	 = detect_axisNumber_0.axis_number;
		choose_attack_mode_0.before_position = before_position;
		choose_attack_mode_0.behind_position = behind_position;
		choose_attack_mode(&choose_attack_mode_0);

		if((choose_attack_mode_0.mode == 1) && (stand_mode == 1)){
			ch_aM->attack_mode = 1; // attack mode If ball is behind of dummy
		}else if((choose_attack_mode_0.mode == 1) && (stand_mode == 2)){
			ch_aM->attack_mode = 2; // attack mode If ball is before of dummy
		}else{
			ch_aM->attack_mode = 0; // If ball it isn't near of dummy
		}

		ch_aM->index_ofAxis = detect_axisNumber_0.axis_number;
	}else{
		ch_aM->attack_mode  = 0;
		ch_aM->index_ofAxis = 0;
	}

}

void detect_axisNumber(struct detect_axisNumber* d_aN)
{
	INT x_posOfD[4];
	REAL x_pos[2];
	USINT i_dAn, a_n[2];

	x_posOfD[0] = 800;
	x_posOfD[1] = 2300;
	x_posOfD[2] = 5300;
	x_posOfD[3] = 8300;

	x_pos[0] = d_aN->ball1_x;
	x_pos[1] = d_aN->ball2_x;

	for(i_dAn = 0; i_dAn < (int)(sizeof(x_pos)/sizeof(x_pos[0])); i_dAn++){
		if(x_pos[i_dAn] >= (x_posOfD[3] - 90)){
			a_n[i_dAn] = 3;
		}else if((x_pos[i_dAn] >= (x_posOfD[2] - 90)) && (x_pos[i_dAn] <= (x_posOfD[3] - 90))){
			a_n[i_dAn] = 2;
		}else if((x_pos[i_dAn] >= (x_posOfD[1] - 90)) && (x_pos[i_dAn] <= (x_posOfD[2] - 90))){
			a_n[i_dAn] = 1;
		}else if((x_pos[i_dAn] >= (x_posOfD[0] - 90)) && (x_pos[i_dAn] <= (x_posOfD[1] - 90))){
			a_n[i_dAn] = 0;
		}else{
			a_n[i_dAn] = 10;
		}

	}

	if((a_n[0] == a_n[1]) || isnan(x_pos[1])){
		d_aN->axis_number = a_n[0];
	}else{
		d_aN->axis_number = a_n[1];
	}
}

void choose_attack_mode(struct choose_attack_mode* ch_aMode)
{
	USINT aux_mode;
	USINT i_df, i_md, i_fw;
	INT x_posOfD[4];
	REAL gk_pos, df_pos[2], md_pos[5], fw_pos[3];

	// auxiliary mode
	aux_mode = 0;
	// initial x pos of axes CPU
	x_posOfD[0] = 800;
	x_posOfD[1] = 2300;
	x_posOfD[2] = 5300;
	x_posOfD[3] = 8300;

	// goalkeeper
	gk_pos = ch_aMode->actual_positionsOfDummies[0];
	// defender
	df_pos[0] = ch_aMode->actual_positionsOfDummies[1];
	df_pos[1] = ch_aMode->actual_positionsOfDummies[2];
	// midfielder
	md_pos[0] = ch_aMode->actual_positionsOfDummies[3];
	md_pos[1] = ch_aMode->actual_positionsOfDummies[4];
	md_pos[2] = ch_aMode->actual_positionsOfDummies[5];
	md_pos[3] = ch_aMode->actual_positionsOfDummies[6];
	md_pos[4] = ch_aMode->actual_positionsOfDummies[7];
	// forward
	fw_pos[0] = ch_aMode->actual_positionsOfDummies[8];
	fw_pos[1] = ch_aMode->actual_positionsOfDummies[9];
	fw_pos[2] = ch_aMode->actual_positionsOfDummies[10];

	switch(ch_aMode->axis_number){
		case 0:
			{
				if((((ch_aMode->ball1_x <= (x_posOfD[ch_aMode->axis_number] + ch_aMode->before_position))
					&& (ch_aMode->ball1_x >= (x_posOfD[ch_aMode->axis_number] + ch_aMode->behind_position)))
					|| ((ch_aMode->ball2_x <= (x_posOfD[ch_aMode->axis_number] + ch_aMode->before_position))
					&& (ch_aMode->ball2_x >= (x_posOfD[ch_aMode->axis_number] + ch_aMode->behind_position))))
					&& ((ch_aMode->ball1_y <= (gk_pos + 150)) && (ch_aMode->ball1_y >= (gk_pos - 150))
					|| ((ch_aMode->ball2_y <= (gk_pos + 150)) && (ch_aMode->ball2_y >= (gk_pos - 150))))){
					aux_mode = 1;
				}else{
					aux_mode = 0;
				}
			}
			break;
		case 1:
			{
				for(i_df = 0; i_df < (int)(sizeof(df_pos)/sizeof(df_pos[0])); i_df++){
					if((((ch_aMode->ball1_x <= (x_posOfD[ch_aMode->axis_number] + ch_aMode->before_position))
						&& (ch_aMode->ball1_x >= (x_posOfD[ch_aMode->axis_number] + ch_aMode->behind_position)))
						|| ((ch_aMode->ball2_x <= (x_posOfD[ch_aMode->axis_number] + ch_aMode->before_position))
						&& (ch_aMode->ball2_x >= (x_posOfD[ch_aMode->axis_number] + ch_aMode->behind_position))))
						&& ((ch_aMode->ball1_y <= (df_pos[i_df] + 150)) && (ch_aMode->ball1_y >= (df_pos[i_df] - 150))
						|| ((ch_aMode->ball2_y <= (df_pos[i_df] + 150)) && (ch_aMode->ball2_y >= (df_pos[i_df] - 150))))){
						aux_mode = 1;
					}
				}
			}
			break;
		case 2:
			{
				for(i_md = 0; i_md < (int)(sizeof(md_pos)/sizeof(md_pos[0])); i_md++){
					if((((ch_aMode->ball1_x <= (x_posOfD[ch_aMode->axis_number] + ch_aMode->before_position))
						&& (ch_aMode->ball1_x >= (x_posOfD[ch_aMode->axis_number] + ch_aMode->behind_position)))
						|| ((ch_aMode->ball2_x <= (x_posOfD[ch_aMode->axis_number] + ch_aMode->before_position))
						&& (ch_aMode->ball2_x >= (x_posOfD[ch_aMode->axis_number] + ch_aMode->behind_position))))
						&& ((ch_aMode->ball1_y <= (md_pos[i_md] + 150)) && (ch_aMode->ball1_y >= (md_pos[i_md] - 150))
						|| ((ch_aMode->ball2_y <= (md_pos[i_md] + 150)) && (ch_aMode->ball2_y >= (md_pos[i_md] - 150))))){
						aux_mode = 1;
					}
				}
			}
			break;
		case 3:
			{
				for(i_fw = 0; i_fw < (int)(sizeof(fw_pos)/sizeof(fw_pos[0])); i_fw++){
					if((((ch_aMode->ball1_x <= (x_posOfD[ch_aMode->axis_number] + ch_aMode->before_position))
						&& (ch_aMode->ball1_x >= (x_posOfD[ch_aMode->axis_number] + ch_aMode->behind_position)))
						|| ((ch_aMode->ball2_x <= (x_posOfD[ch_aMode->axis_number] + ch_aMode->before_position))
						&& (ch_aMode->ball2_x >= (x_posOfD[ch_aMode->axis_number] + ch_aMode->behind_position))))
						&& ((ch_aMode->ball1_y <= (fw_pos[i_fw] + 150)) && (ch_aMode->ball1_y >= (fw_pos[i_fw] - 150))
						|| ((ch_aMode->ball2_y <= (fw_pos[i_fw] + 150)) && (ch_aMode->ball2_y >= (fw_pos[i_fw] - 150))))){
						aux_mode = 1;
					}
				}
			}
			break;
	}// end switch

	if(aux_mode == 1){
		ch_aMode->mode = aux_mode;
	}else{
		ch_aMode->mode = 0;
	}
}
```

#### axes_control.c
```c
#include <bur/plctypes.h>
#include <stdio.h>
#include <stdlib.h>
#include <MpAxis.h>

#ifdef __cplusplus
	extern "C"
	{
#endif
	#include "rp_funcx1.h"
#ifdef __cplusplus
	};
#endif
void init_control_axis(struct axes_control* a_c);

void axes_control(struct axes_control* a_c)
{

	if(!a_c->Enable){
		init_control_axis(&a_c);
	}

	switch(a_c->Internal.state){
		case 0:
			{
				a_c->Internal.before_state = 0;

				if(a_c->start_move == 1){
					a_c->successfully = 0;
					if(((a_c->rotary_axis_cyclic->Error == 1 && a_c->rotary_axis_cyclic->StatusID != 0) || (a_c->linear_axis_cyclic->Error == 1 && a_c->linear_axis_cyclic->StatusID != 0))
					|| (a_c->rotary_axis_cyclic->CommandAborted == 1 || a_c->linear_axis_cyclic->CommandAborted == 1)){
						// cyclic position -> off
						a_c->linear_axis_cyclic->CyclicPosition = 0;
						a_c->rotary_axis_cyclic->CyclicPosition = 0;
						if(a_c->linear_axis_cyclic->CyclicPosition == 0 && a_c->rotary_axis_cyclic->CyclicPosition == 0){
							// go to error state
							a_c->Internal.state = 10;
						}
					}else{
						// start cyclic position
						a_c->linear_axis_cyclic->CyclicPosition = 1;
						a_c->rotary_axis_cyclic->CyclicPosition = 1;
						// go to next state
						a_c->Internal.state = 1;
					}
				}else if(((a_c->rotary_axis_cyclic->Error == 1 && a_c->rotary_axis_cyclic->StatusID != 0) || (a_c->linear_axis_cyclic->Error == 1 && a_c->linear_axis_cyclic->StatusID != 0))
				|| (a_c->rotary_axis_cyclic->CommandAborted == 1 || a_c->linear_axis_cyclic->CommandAborted == 1)){
					// cyclic position -> off
					a_c->linear_axis_cyclic->CyclicPosition = 0;
					a_c->rotary_axis_cyclic->CyclicPosition = 0;
					if(a_c->linear_axis_cyclic->CyclicPosition == 0 && a_c->rotary_axis_cyclic->CyclicPosition == 0){
						// go to error state
						a_c->Internal.state = 10;
					}
				}
			}
			break;
		case 1:
			{
				a_c->Internal.before_state = 1;

				if(a_c->linear_axis_param->Acceleration == a_c->linear_param.acceleration && a_c->linear_axis_cyclic->Velocity == a_c->linear_param.velocity){
					if(a_c->rotary_axis_param->Acceleration == a_c->rotary_param.acceleration && a_c->rotary_axis_cyclic->Velocity == a_c->rotary_param.velocity){
						if(((a_c->rotary_axis_cyclic->Error == 1 && a_c->rotary_axis_cyclic->StatusID != 0) || (a_c->linear_axis_cyclic->Error == 1 && a_c->linear_axis_cyclic->StatusID != 0))
						|| (a_c->rotary_axis_cyclic->CommandAborted == 1 || a_c->linear_axis_cyclic->CommandAborted == 1)){
							// cyclic position -> off
							a_c->linear_axis_cyclic->CyclicPosition = 0;
							a_c->rotary_axis_cyclic->CyclicPosition = 0;
							if(a_c->linear_axis_cyclic->CyclicPosition == 0 && a_c->rotary_axis_cyclic->CyclicPosition == 0){
								// go to error state
								a_c->Internal.state = 10;
							}
						}else{
							a_c->Internal.state = 2;
						}
					}else{
						if(((a_c->rotary_axis_cyclic->Error == 1 && a_c->rotary_axis_cyclic->StatusID != 0) || (a_c->linear_axis_cyclic->Error == 1 && a_c->linear_axis_cyclic->StatusID != 0))
						|| (a_c->rotary_axis_cyclic->CommandAborted == 1 || a_c->linear_axis_cyclic->CommandAborted == 1)){
							// cyclic position -> off
							a_c->linear_axis_cyclic->CyclicPosition = 0;
							a_c->rotary_axis_cyclic->CyclicPosition = 0;
							if(a_c->linear_axis_cyclic->CyclicPosition == 0 && a_c->rotary_axis_cyclic->CyclicPosition == 0){
								// go to error state
								a_c->Internal.state = 10;
							}
						}else{
							a_c->Internal.state = 3;
						}
					}
				}else{
					if(a_c->rotary_axis_param->Acceleration == a_c->rotary_param.acceleration && a_c->rotary_axis_cyclic->Velocity == a_c->rotary_param.velocity){
						if(((a_c->rotary_axis_cyclic->Error == 1 && a_c->rotary_axis_cyclic->StatusID != 0) || (a_c->linear_axis_cyclic->Error == 1 && a_c->linear_axis_cyclic->StatusID != 0))
						|| (a_c->rotary_axis_cyclic->CommandAborted == 1 || a_c->linear_axis_cyclic->CommandAborted == 1)){
							// cyclic position -> off
							a_c->linear_axis_cyclic->CyclicPosition = 0;
							a_c->rotary_axis_cyclic->CyclicPosition = 0;
							if(a_c->linear_axis_cyclic->CyclicPosition == 0 && a_c->rotary_axis_cyclic->CyclicPosition == 0){
								// go to error state
								a_c->Internal.state = 10;
							}
						}else{
							a_c->Internal.state = 4;
						}
					}else{
						if(((a_c->rotary_axis_cyclic->Error == 1 && a_c->rotary_axis_cyclic->StatusID != 0) || (a_c->linear_axis_cyclic->Error == 1 && a_c->linear_axis_cyclic->StatusID != 0))
						|| (a_c->rotary_axis_cyclic->CommandAborted == 1 || a_c->linear_axis_cyclic->CommandAborted == 1)){
							// cyclic position -> off
							a_c->linear_axis_cyclic->CyclicPosition = 0;
							a_c->rotary_axis_cyclic->CyclicPosition = 0;
							if(a_c->linear_axis_cyclic->CyclicPosition == 0 && a_c->rotary_axis_cyclic->CyclicPosition == 0){
								// go to error state
								a_c->Internal.state = 10;
							}
						}else{
							a_c->Internal.state = 5;
						}
					}
				}
			}
			break;
		case 2:
			{
				a_c->Internal.before_state = 2;

				// linear axis param cyclic
				a_c->linear_axis_cyclic->Position 				= a_c->linear_param.displacement;
				// rotary axis param cyclic
				a_c->rotary_axis_cyclic->Position 				= a_c->rotary_param.displacement;

				if(((a_c->rotary_axis_cyclic->Error == 1 && a_c->rotary_axis_cyclic->StatusID != 0) || (a_c->linear_axis_cyclic->Error == 1 && a_c->linear_axis_cyclic->StatusID != 0))
				|| (a_c->rotary_axis_cyclic->CommandAborted == 1 || a_c->linear_axis_cyclic->CommandAborted == 1)){
					// cyclic position -> off
					a_c->linear_axis_cyclic->CyclicPosition = 0;
					a_c->rotary_axis_cyclic->CyclicPosition = 0;
					if(a_c->linear_axis_cyclic->CyclicPosition == 0 && a_c->rotary_axis_cyclic->CyclicPosition == 0){
						// go to error state
						a_c->Internal.state = 10;
					}
				}else{
					a_c->Internal.state = 6;
				}
			}
			break;
		case 3:
			{
				a_c->Internal.before_state = 3;
				// turn off
				a_c->rotary_axis_cyclic->CyclicPosition = 0;

				if(a_c->rotary_axis_cyclic->CyclicPosition == 0){
					// linear axis param cyclic
					a_c->linear_axis_cyclic->Velocity   			= a_c->linear_param.velocity;
					a_c->linear_axis_cyclic->Position 				= a_c->linear_param.displacement;
					// rotary axis param
					a_c->rotary_axis_param->Acceleration		    = a_c->rotary_param.acceleration;
					a_c->rotary_axis_param->Deceleration			= a_c->rotary_param.deceleration;
					// rotary axis param cyclic
					a_c->rotary_axis_cyclic->Velocity   			= a_c->rotary_param.velocity;
					a_c->rotary_axis_cyclic->Position 				= a_c->rotary_param.displacement;

					// update parameters
					a_c->rotary_axis_cyclic->Update = 1;

					if(((a_c->rotary_axis_cyclic->Error == 1 && a_c->rotary_axis_cyclic->StatusID != 0) || (a_c->linear_axis_cyclic->Error == 1 && a_c->linear_axis_cyclic->StatusID != 0))
					 || (a_c->rotary_axis_cyclic->CommandAborted == 1 || a_c->linear_axis_cyclic->CommandAborted == 1)){
						// cyclic position -> off
						a_c->linear_axis_cyclic->CyclicPosition = 0;
						a_c->rotary_axis_cyclic->CyclicPosition = 0;
						if(a_c->linear_axis_cyclic->CyclicPosition == 0 && a_c->rotary_axis_cyclic->CyclicPosition == 0){
							// go to error state
							a_c->Internal.state = 10;
						}
					}else{
						if(a_c->rotary_axis_cyclic->UpdateDone == 1){
							a_c->rotary_axis_cyclic->Update = 0;
							if(a_c->rotary_axis_cyclic->Update == 0){
								// turn on
								a_c->rotary_axis_cyclic->CyclicPosition = 1;
								if(a_c->rotary_axis_cyclic->CyclicPosition == 1){
									a_c->Internal.state = 6;
								}
							}
						}
					}
				}
			}
			break;
		case 4:
			{
				a_c->Internal.before_state = 4;

				// turn off
				a_c->linear_axis_cyclic->CyclicPosition = 0;

				if(a_c->linear_axis_cyclic->CyclicPosition == 0){
					// linear axis param
					a_c->linear_axis_param->Acceleration		    = a_c->linear_param.acceleration;
					a_c->linear_axis_param->Deceleration			= a_c->linear_param.deceleration;
					// linear axis param cyclic
					a_c->linear_axis_cyclic->Velocity   			= a_c->linear_param.velocity;
					a_c->linear_axis_cyclic->Position 				= a_c->linear_param.displacement;
					// rotary axis param cyclic
					a_c->rotary_axis_cyclic->Velocity   			= a_c->rotary_param.velocity;
					a_c->rotary_axis_cyclic->Position 				= a_c->rotary_param.displacement;

					// update parameters
					a_c->linear_axis_cyclic->Update = 1;

					if(((a_c->rotary_axis_cyclic->Error == 1 && a_c->rotary_axis_cyclic->StatusID != 0) || (a_c->linear_axis_cyclic->Error == 1 && a_c->linear_axis_cyclic->StatusID != 0))
					|| (a_c->rotary_axis_cyclic->CommandAborted == 1 || a_c->linear_axis_cyclic->CommandAborted == 1)){
						// cyclic position -> off
						a_c->linear_axis_cyclic->CyclicPosition = 0;
						a_c->rotary_axis_cyclic->CyclicPosition = 0;
						if(a_c->linear_axis_cyclic->CyclicPosition == 0 && a_c->rotary_axis_cyclic->CyclicPosition == 0){
							// go to error state
							a_c->Internal.state = 10;
						}
					}else{
						if(a_c->linear_axis_cyclic->UpdateDone == 1){
							a_c->linear_axis_cyclic->Update = 0;
							if(a_c->linear_axis_cyclic->Update == 0){
								// turn on
								a_c->linear_axis_cyclic->CyclicPosition = 1;
								if(a_c->linear_axis_cyclic->CyclicPosition == 1){
									a_c->Internal.state = 6;
								}
							}
						}
					}
				}
			}
			break;
		case 5:
			{
				a_c->Internal.before_state = 5;

				// turn off
				a_c->linear_axis_cyclic->CyclicPosition = 0;
				a_c->rotary_axis_cyclic->CyclicPosition = 0;

				if(a_c->linear_axis_cyclic->CyclicPosition == 0 && a_c->rotary_axis_cyclic->CyclicPosition == 0){
					// linear axis param
					a_c->linear_axis_param->Acceleration		    = a_c->linear_param.acceleration;
					a_c->linear_axis_param->Deceleration			= a_c->linear_param.deceleration;
					// linear axis param cyclic
					a_c->linear_axis_cyclic->Velocity   			= a_c->linear_param.velocity;
					a_c->linear_axis_cyclic->Position 				= a_c->linear_param.displacement;
					// rotary axis param
					a_c->rotary_axis_param->Acceleration		    = a_c->rotary_param.acceleration;
					a_c->rotary_axis_param->Deceleration			= a_c->rotary_param.deceleration;
					// rotary axis param cyclic
					a_c->rotary_axis_cyclic->Velocity   			= a_c->rotary_param.velocity;
					a_c->rotary_axis_cyclic->Position 				= a_c->rotary_param.displacement;

					// update parameters
					a_c->linear_axis_cyclic->Update = 1;
					a_c->rotary_axis_cyclic->Update = 1;

					if(((a_c->rotary_axis_cyclic->Error == 1 && a_c->rotary_axis_cyclic->StatusID != 0) || (a_c->linear_axis_cyclic->Error == 1 && a_c->linear_axis_cyclic->StatusID != 0))
					|| (a_c->rotary_axis_cyclic->CommandAborted == 1 || a_c->linear_axis_cyclic->CommandAborted == 1)){
						// cyclic position -> off
						a_c->linear_axis_cyclic->CyclicPosition = 0;
						a_c->rotary_axis_cyclic->CyclicPosition = 0;
						if(a_c->linear_axis_cyclic->CyclicPosition == 0 && a_c->rotary_axis_cyclic->CyclicPosition == 0){
							// go to error state
							a_c->Internal.state = 10;
						}
					}else{
						if(a_c->linear_axis_cyclic->UpdateDone == 1 && a_c->rotary_axis_cyclic->UpdateDone == 1){
							a_c->linear_axis_cyclic->Update = 0;
							a_c->rotary_axis_cyclic->Update = 0;
							if(a_c->linear_axis_cyclic->Update == 0 && a_c->rotary_axis_cyclic->Update == 0){
								// turn on
								a_c->linear_axis_cyclic->CyclicPosition = 1;
								a_c->rotary_axis_cyclic->CyclicPosition = 1;
								if(a_c->linear_axis_cyclic->CyclicPosition == 1 && a_c->rotary_axis_cyclic->CyclicPosition == 1){
									a_c->Internal.state = 6;
								}
							}
						}
					}
				}
			}
			break;
		case 6:
			{
				a_c->Internal.before_state = 6;

				if(((a_c->rotary_axis_cyclic->Error == 1 && a_c->rotary_axis_cyclic->StatusID != 0) || (a_c->linear_axis_cyclic->Error == 1 && a_c->linear_axis_cyclic->StatusID != 0))
				|| (a_c->rotary_axis_cyclic->CommandAborted == 1 || a_c->linear_axis_cyclic->CommandAborted == 1)){
					// cyclic position -> off
					a_c->linear_axis_cyclic->CyclicPosition = 0;
					a_c->rotary_axis_cyclic->CyclicPosition = 0;
					if(a_c->linear_axis_cyclic->CyclicPosition == 0 && a_c->rotary_axis_cyclic->CyclicPosition == 0){
						// go to error state
						a_c->Internal.state = 10;
					}
				}else{
					a_c->successfully = 1;

					if(a_c->successfully == 1){
						a_c->Internal.state = 0;
					}
				}
			}
			break;
		case 10:
			{
				// error reset -> on
				a_c->rotary_axis_cyclic->ErrorReset = 1;
				a_c->linear_axis_cyclic->ErrorReset = 1;

				if((a_c->rotary_axis_cyclic->Error == 0 && a_c->linear_axis_cyclic->Error == 0 && a_c->rotary_axis_cyclic->StatusID == 0 && a_c->linear_axis_cyclic->StatusID == 0)
				&& (a_c->rotary_axis_cyclic->CommandAborted == 0 && a_c->linear_axis_cyclic->CommandAborted == 0)){
					// error reset -> off
					a_c->rotary_axis_cyclic->ErrorReset = 0;
					a_c->linear_axis_cyclic->ErrorReset = 0;
					// cyclic position -> on
					a_c->linear_axis_cyclic->CyclicPosition = 1;
					a_c->rotary_axis_cyclic->CyclicPosition = 1;

					if(a_c->rotary_axis_cyclic->ErrorReset == 0 && a_c->linear_axis_cyclic->ErrorReset == 0){
						a_c->Internal.state = a_c->Internal.before_state;
					}
				}

			}
			break;
	}// end switch

}// end function

void init_control_axis(struct axes_control* a_c)
{
	a_c->Internal.state 	   = 0;
	a_c->Internal.before_state = 0;
	a_c->successfully 		   = 0;
}
```

#### calculation_posDummiesOpponent.c - not listed in the package file held
```c
/*********************************************************************************************
* B&R Automation - Perfection in Automation (https://www.br-automation.com)
    ******************************************************************************************
    * Program 	    : Master's Thesis - Soccer Table (Simulation)
    * Author  	    : Roman Parak
    * Created 	    : date ...
	* University    : Brno University of Technology(BUT)
	* Faculty       : Faculty of Mechanical Engineering(FME)
	* Study Program : Applied Computer Science and Control
	* Institute     : Institute of Automation and Computer Science
**********************************************************************************************
* Implementation OF PROGRAM simulation(rp_library/rp_funcx1/calculation_posDummiesOpponent.c)
**********************************************************************************************/

/************************************* LIBRARIES *********************************************/
#include <bur/plctypes.h>
#ifdef __cplusplus
	extern "C"
	{
#endif
	#include "rp_funcx1.h"
#ifdef __cplusplus
	};
#endif

/**********************************************************************************************************/
/************************************** FUNCTIONS & FUNCTIONS BLOCKS **************************************/
/**********************************************************************************************************/

void calculation_posDummiesOpponent(struct calculation_posDummiesOpponent* c_pD)
{
	/*
		Args:
			INPUT
				displacement_HUMAN : displacement of individual axes(HUMAN)a
								     array of data type REAL, where the index of array is individual axis
								     e.g. goalkeeper has index 0 etc.
			OUTPUT
				gk_posD 		   : position dummy of the axis name Goalkeeper
									 1 position
				df_posD 		   : position dummies of the axis name Defender
									 2 positions
				md_posD 		   : position dummies of the axis name Midfielder
									 5 positions
				fw_posD 		   : position dummies of the axis name Forward
									 3 positions
				real_displacement  : real displacement, for example due to mistake at reading from the sensors
									 array of data type REAL - all output values
	*/

	/***************************************** declaration variables ****************************************/
	REAL max_dispOfD[4], min_dispOfD[4], matrix_posOfOpponent[4][5], actual_positions[4][5];
	USINT i,j;
	// Indexes : GK - 0, DF - 1, MD - 2, FW - 3
	// max displacement of dummies
	max_dispOfD[0] = 1000;
	max_dispOfD[1] = 1850;
	max_dispOfD[2] = 650;
	max_dispOfD[3] = 955;
	// min displacement of dummies
	min_dispOfD[0] = -1000;
	min_dispOfD[1] = -1850;
	min_dispOfD[2] = -650;
	min_dispOfD[3] = -955;
	// matrix of parameters
	// goalkeeper
	matrix_posOfOpponent[0][0] = 0;
	// defender
	matrix_posOfOpponent[1][0] = -1200;
	matrix_posOfOpponent[1][1] = 1200;
	// midfielder
	matrix_posOfOpponent[2][0] = -2400;
	matrix_posOfOpponent[2][1] = -1200;
	matrix_posOfOpponent[2][2] = 0;
	matrix_posOfOpponent[2][3] = 1200;
	matrix_posOfOpponent[2][4] = 2400;
	// forward
	matrix_posOfOpponent[3][0] = -2100;
	matrix_posOfOpponent[3][1] = 0;
	matrix_posOfOpponent[3][2] = 2100;

	/********************************************* calculation **********************************************/
	for(i = 0; i < (int)(sizeof(c_pD->displacement_HUMAN)/sizeof(c_pD->displacement_HUMAN[0])); i++){
		for(j = 0; j <= (int)(sizeof(c_pD->displacement_HUMAN)/sizeof(c_pD->displacement_HUMAN[0])); j++){
			if(c_pD->displacement_HUMAN[i] > max_dispOfD[i]){
				actual_positions[i][j] 	   = max_dispOfD[i] + matrix_posOfOpponent[i][j];
				c_pD->real_displacement[i] = max_dispOfD[i];
			}else if(c_pD->displacement_HUMAN[i] < min_dispOfD[i]){
				actual_positions[i][j] 	   = min_dispOfD[i] + matrix_posOfOpponent[i][j];
				c_pD->real_displacement[i] = min_dispOfD[i];
			}else{
				actual_positions[i][j]     = c_pD->displacement_HUMAN[i] + matrix_posOfOpponent[i][j];
				c_pD->real_displacement[i] = c_pD->displacement_HUMAN[i];
			}
		}
	}

	/**************************************** output real parameters ****************************************/
	// goalkeeper
	c_pD->gk_posD    = actual_positions[0][0];
	// defender
	c_pD->df_posD[0] = actual_positions[1][0];
	c_pD->df_posD[1] = actual_positions[1][1];
	// midfielder
	c_pD->md_posD[0] = actual_positions[2][0];
	c_pD->md_posD[1] = actual_positions[2][1];
	c_pD->md_posD[2] = actual_positions[2][2];
	c_pD->md_posD[3] = actual_positions[2][3];
	c_pD->md_posD[4] = actual_positions[2][4];
	// forward
	c_pD->fw_posD[0] = actual_positions[3][0];
	c_pD->fw_posD[1] = actual_positions[3][1];
	c_pD->fw_posD[2] = actual_positions[3][2];

}// end function
```

#### powerOn_axes.c - not listed in the package file held
```c
#include <bur/plctypes.h>
#include <stdio.h>
#include <stdlib.h>
#include <MpAxis.h>

#ifdef __cplusplus
	extern "C"
	{
#endif
	#include "rp_funcx1.h"
#ifdef __cplusplus
	};
#endif
void initialization_pO_a(struct powerOn_axes* pO_a);

void powerOn_axes(struct powerOn_axes* pO_a)
{
	if(!pO_a->start_btn){
		initialization_pO_a(pO_a);
	}

	switch(pO_a->Internal.state){
		case 0:
			{
				pO_a->Internal.before_state     = pO_a->Internal.state;

				if(pO_a->axis_name_R->Error == 1 || pO_a->axis_name_R->StatusID != 0 || pO_a->axis_name_L->Error == 1 || pO_a->axis_name_L->StatusID != 0){
					pO_a->Internal.state = 10;
				}else{
					if(pO_a->start_btn == 1){
						pO_a->Internal.state = 1;
					}
				}
			}
			break;
		case 1:
			{
				pO_a->Internal.before_state = pO_a->Internal.state;
				// power on -> axis
				pO_a->axis_name_R->Power = 1;
				pO_a->axis_name_L->Power = 1;

				if(pO_a->axis_name_R->PowerOn == 1 && pO_a->axis_name_L->PowerOn == 1){
					pO_a->succesfully = 1;
				}else if(pO_a->axis_name_R->Error == 1 || pO_a->axis_name_L->StatusID != 0){
					pO_a->Internal.state = 10;
				}else{
					pO_a->Internal.state = pO_a->Internal.before_state;
				}
			}
			break;
		case 10:
			{
				pO_a->axis_name_R->ErrorReset = 1;
				pO_a->axis_name_L->ErrorReset = 1;

			if(pO_a->axis_name_R->Error == 1 || pO_a->axis_name_R->StatusID != 0 || pO_a->axis_name_L->Error == 1 || pO_a->axis_name_L->StatusID != 0){
					pO_a->Internal.state = 10;
				}else{
					pO_a->axis_name_R->ErrorReset = 0;
					pO_a->axis_name_L->ErrorReset = 0;
					pO_a->Internal.state 		= pO_a->Internal.before_state;
				}
			}
			break;
	}// end switch
}// end function

void initialization_pO_a(struct powerOn_axes* pO_a)
{
	pO_a->Internal.state 		= 0;
	pO_a->Internal.before_state = 0;
	pO_a->start_btn				= 0;
	pO_a->succesfully     		= 0;
}// end function
```

#### test.c - not listed in the package file held
```c
#include <bur/plctypes.h>
#include <stdio.h>
#include <stdlib.h>
#include <MpAxis.h>

#ifdef __cplusplus
	extern "C"
	{
#endif
	#include "rp_funcx1.h"
#ifdef __cplusplus
	};
#endif
/* TODO: Add your comment here */
void test(struct test* inst)
{
	inst->b = inst->a->Active;
}
```

### Package Logical/Libraries/RO_LB_ScoreDetection - Lubo and Radek Library for detection of score.

- Library Logical/Libraries/RO_LB_ScoreDetection/Scorkeeper (ANSIC) (no source held here)

### Library Logical/Libraries/RO_LB_ScoreDetection/GoalKeeper

#### Types.typ
```iecst
TYPE
	DI9371_type : 	STRUCT
		ModuleOk : BOOL;
		DigitalInput : BOOL;
	END_STRUCT;
	InternalG_type : 	STRUCT
		init : BOOL;
		DisableTimer : TON_10ms;
	END_STRUCT;
	MappViewG_type : 	STRUCT
		counter : INT;
	END_STRUCT;
END_TYPE
```

#### GoalKeeper.fun
```iecst
FUNCTION_BLOCK GoalKeeper
	VAR_INPUT
		enable : BOOL;
		DI9371 : DI9371_type;
	END_VAR
	VAR_OUTPUT
		status : UINT;
		isGoal : BOOL;
	END_VAR
	VAR
		MappView : MappViewG_type;
		Internal : InternalG_type;
	END_VAR
END_FUNCTION_BLOCK
```

#### GoalKeeper.c
```c
#include <bur/plctypes.h>

#ifdef _DEFAULT_INCLUDES
#include <AsDefault.h>
#endif

void GoalKeeper(struct GoalKeeper *inst){

	if (inst->enable){
		if (!inst->Internal.init){
			inst->Internal.DisableTimer.PT = 500;
			inst->Internal.init = 1;
		}

		if (!inst->DI9371.ModuleOk)
			inst->status = ERR_DI_NOTFOUND;
		else
			inst->status = ERR_OK;

		TON_10ms(&inst->Internal.DisableTimer);

		if ((inst->Internal.DisableTimer.IN == 1) && (inst->Internal.DisableTimer.Q)){
			inst->Internal.DisableTimer.IN = 0;
		}
		else if ((!inst->DI9371.DigitalInput) && (!inst->isGoal) && (!inst->Internal.DisableTimer.IN)) {
			inst->isGoal = 1;
			inst->MappView.counter = inst->MappView.counter + 1;
			inst->Internal.DisableTimer.IN = 1;
		}
		else{
				inst->isGoal = 0;
			}
	}
	else
		inst->status = ERR_FUB_ENABLE_FALSE;
}
```

### Library Logical/Libraries/RO_Sensors/Library (IEC)

#### Types.typ - Exported data types
```iecst
TYPE
	PositionStatus :
		(
		PosCalcPos, (*1*)
		PosInitial
		);
	Stuct_OptSensInternal : 	STRUCT
		Index : ARRAY[0..4]OF USINT;
		DetRot_ModulOK_0 : DetectionRotation;
		DetPos_Figure_0 : DetPos_Figure;
		MinAccDiff : INT := 100;
		MaxAccDiff : ARRAY[0..3]OF INT := [4(100)];
		CurrentPosition : ARRAY[0..3]OF INT;
	END_STRUCT;
	Stuct_RexlSensInternal : 	STRUCT
		IndexR : ARRAY[0..1]OF USINT;
	END_STRUCT;
END_TYPE
```

#### Library.fun - Exported functions and function blocks
```iecst
FUNCTION_BLOCK DetectionPositionAxis
	VAR_INPUT
		ActPosSens : ARRAY[0..3] OF INT;
		ErrorOptSens : ARRAY[0..3] OF BOOL;
		ModulOK : ARRAY[0..3] OF BOOL;
	END_VAR
	VAR_OUTPUT
		ActPosHumFig : ARRAY[0..10] OF INT;
		ActPosHumAxis : ARRAY[0..3] OF INT;
		ExternalModulOK : ARRAY[0..3] OF BOOL;
	END_VAR
	VAR CONSTANT
		RefPosSens : ARRAY[0..3] OF INT := [4(0)];
		MaxPosSens : ARRAY[0..3] OF INT := [4(0)];
		MinPosSens : ARRAY[0..3] OF INT := [4(0)];
		RefPosHum : ARRAY[0..3] OF INT := [4(0)];
		MaxPosHum : ARRAY[0..3] OF INT := [4(0)];
		MinPosHum : ARRAY[0..3] OF INT := [4(0)];
	END_VAR
	VAR
		TransConst : ARRAY[0..3] OF INT;
		InternalPos : Stuct_OptSensInternal;
	END_VAR
END_FUNCTION_BLOCK

FUNCTION_BLOCK DetectionRotation
	VAR_OUTPUT
		ExternalModulRotOK : ARRAY[0..3] OF BOOL;
	END_VAR
	VAR_INPUT
		ErrorReflSens : ARRAY[0..3] OF BOOL;
		ModulRotOK : ARRAY[0..3] OF BOOL;
	END_VAR
	VAR_OUTPUT
		ActReflRotOP : ARRAY[0..3] OF BOOL;
	END_VAR
	VAR
		InternalRot : Stuct_RexlSensInternal;
	END_VAR
END_FUNCTION_BLOCK

FUNCTION_BLOCK DetPos_Figure
	VAR_INPUT
		ActPosHumAxisDP : ARRAY[0..3] OF INT;
	END_VAR
	VAR_OUTPUT
		ActPosHumFigDP : ARRAY[0..10] OF INT;
	END_VAR
	VAR
		DispAxisDP : ARRAY[0..10] OF INT := [11(0)];
		i1 : USINT;
		i2 : USINT;
		i3 : USINT;
		MaxPosHumDP : ARRAY[0..3] OF INT := [4(0)];
		MinPosHumDP : ARRAY[0..3] OF INT := [4(0)];
	END_VAR
END_FUNCTION_BLOCK
```

#### DetectionRotation.st
```iecst
(* LOGIC PREDICTION OF ROTATION ALL AXES *)
FUNCTION_BLOCK DetectionRotation

	// Set the value of index
	InternalRot.IndexR[0] := 0;

	// Checking the status of reflex sensor
	FOR InternalRot.IndexR[0] := 0 TO 3 DO

		// Reflex sensor works & Modul set TRUE to output
		IF (ModulRotOK[InternalRot.IndexR[0]] = TRUE) AND (ErrorReflSens[InternalRot.IndexR[0]] = FALSE) THEN
			ActReflRotOP[InternalRot.IndexR[0]] := ModulRotOK[InternalRot.IndexR[0]];

		// Reflex sensor works but Modul set FALSE to output
		ELSIF (ModulRotOK[InternalRot.IndexR[0]] = FALSE) AND (ErrorReflSens[InternalRot.IndexR[0]] = FALSE) THEN
				ActReflRotOP[InternalRot.IndexR[0]] := ModulRotOK[InternalRot.IndexR[0]];

			// Reflex sensor doesn't works
		ELSIF (ErrorReflSens[InternalRot.IndexR[0]] = TRUE) THEN
			ActReflRotOP[InternalRot.IndexR[0]] := FALSE;

		// 	Set the status of Actual position of Rotation by the ModulOK status
		ELSE
			ActReflRotOP[InternalRot.IndexR[0]] := ModulRotOK[InternalRot.IndexR[0]];
		END_IF
	END_FOR

END_FUNCTION_BLOCK
```

#### DetectionPositionAxis.st
```iecst
(* NUMERIC CALCULATION OF POSITION ALL AXES *)
FUNCTION_BLOCK DetectionPositionAxis

	// Init part of program set the basic values & constants

		// Reset output variables
		InternalPos.Index[0] := 0;
		InternalPos.Index[1] := 0;
		InternalPos.Index[2] := 0;
		InternalPos.Index[3] := 0;
		InternalPos.Index[4] := 0;

		// Referent positions
		ActPosHumAxis[0] := RefPosHum[0];
		ActPosHumAxis[1] := RefPosHum[1];
		ActPosHumAxis[2] := RefPosHum[2];
		ActPosHumAxis[3] := RefPosHum[3];

		// Previous position
		InternalPos.CurrentPosition[0] := RefPosHum[0];
		InternalPos.CurrentPosition[1] := RefPosHum[1];
		InternalPos.CurrentPosition[2] := RefPosHum[2];
		InternalPos.CurrentPosition[3] := RefPosHum[3];

		// Calculate a constants
		TransConst[0] := (MaxPosSens[0]-MinPosSens[0])/(MaxPosHum[0]-MinPosHum[0]);
		TransConst[1] := (MaxPosSens[1]-MinPosSens[1])/(MaxPosHum[1]-MinPosHum[1]);
		TransConst[2] := (MaxPosSens[2]-MinPosSens[2])/(MaxPosHum[2]-MinPosHum[2]);
		TransConst[3] := (MaxPosSens[3]-MinPosSens[3])/(MaxPosHum[3]-MinPosHum[3]);

		// Status of Reflex sensors (set in position of blocking the ball)
		ModulOK[0] := TRUE;
		ModulOK[1] := TRUE;
		ModulOK[2] := TRUE;
		ModulOK[3] := TRUE;

	// Check the status of Reflex sensors if they work well (TRUE = figure block the balon; FALSE = figure open the way)
	FOR InternalPos.Index[1] := 0 TO 3 DO

		InternalPos.DetRot_ModulOK_0.ModulRotOK[InternalPos.Index[1]] := ModulOK[InternalPos.Index[1]];
		InternalPos.DetRot_ModulOK_0();
		ExternalModulOK[InternalPos.Index[1]] := InternalPos.DetRot_ModulOK_0.ExternalModulRotOK[InternalPos.Index[1]];

	END_FOR;

	// Calculation state compute an atual value of distance or set the max/min value
	FOR InternalPos.Index[0] := 0 TO 3 DO

		// Optical sensor work well and values are in range and diference is over the minimal limit (compute a position by equation)
		IF (ErrorOptSens[InternalPos.Index[0]] = FALSE) AND ((ActPosSens[InternalPos.Index[0]] < MaxPosSens[InternalPos.Index[0]]) AND (ABS(ActPosSens[InternalPos.Index[0]] - InternalPos.CurrentPosition[InternalPos.Index[0]]) > InternalPos.MaxAccDiff[0])) AND ((ActPosSens[InternalPos.Index[0]] > MinPosSens[InternalPos.Index[0]]) AND (ABS(ActPosSens[InternalPos.Index[0]] - InternalPos.CurrentPosition[InternalPos.Index[0]]) > InternalPos.MaxAccDiff[0])) THEN
			ActPosHumAxis[InternalPos.Index[0]] := RefPosHum[InternalPos.Index[0]] + ((ActPosSens[InternalPos.Index[0]] - RefPosSens[InternalPos.Index[0]]) / TransConst[InternalPos.Index[0]]);
			InternalPos.CurrentPosition[InternalPos.Index[0]]:= ActPosHumAxis[InternalPos.Index[0]]; // Last detected value is safed as previous value for case Error mode of sensor

		// Optical sensor work well and values are in range and diference is in the minimal limit (set the previous value of position)
		ELSIF (ErrorOptSens[InternalPos.Index[0]] = FALSE) AND ((ActPosSens[InternalPos.Index[0]] < MaxPosSens[InternalPos.Index[0]]) AND (ABS(ActPosSens[InternalPos.Index[0]] - InternalPos.CurrentPosition[InternalPos.Index[0]]) < InternalPos.MaxAccDiff[0])) AND ((ActPosSens[InternalPos.Index[0]] > MinPosSens[InternalPos.Index[0]]) AND (ABS(ActPosSens[InternalPos.Index[0]] - InternalPos.CurrentPosition[InternalPos.Index[0]]) < InternalPos.MaxAccDiff[0])) THEN
			ActPosHumAxis[InternalPos.Index[0]]	:= InternalPos.CurrentPosition[InternalPos.Index[0]]; // Previous value of position

		// Optical sensor doesn't work well but values are in range
		ELSIF (ErrorOptSens[InternalPos.Index[0]] = TRUE) AND (ActPosSens[InternalPos.Index[0]] < MaxPosSens[InternalPos.Index[0]]) AND (ActPosSens[InternalPos.Index[0]] > MinPosSens[InternalPos.Index[0]]) THEN
			ActPosHumAxis[InternalPos.Index[0]] := 	InternalPos.CurrentPosition[InternalPos.Index[0]]; // Previous value of position

		// Optical sensor doesn't work well but values are over the maximum range
		ELSIF (ErrorOptSens[InternalPos.Index[0]] = TRUE) AND (ActPosSens[InternalPos.Index[0]] > MaxPosSens[InternalPos.Index[0]]) THEN
			ActPosHumAxis[InternalPos.Index[0]] := 	MaxPosSens[InternalPos.Index[0]]; // Maximum value of the range

		// Optical sensor doesn't work well but values are less than the minimum range
		ELSIF (ErrorOptSens[InternalPos.Index[0]] = TRUE) AND (ActPosSens[InternalPos.Index[0]] < MinPosSens[InternalPos.Index[0]]) AND (ActPosSens[InternalPos.Index[0]] > InternalPos.MinAccDiff ) THEN
			ActPosHumAxis[InternalPos.Index[0]] := 	MinPosSens[InternalPos.Index[0]]; // Minimum value of the range

		// Check if the Optical sensors are switched on (if not, sensored values are in range <-5 ; +5> _ the minimum limit sets InternalPos.MinAccDiff)
		ELSIF (ActPosSens[InternalPos.Index[0]] < InternalPos.MinAccDiff) THEN
			ActPosHumAxis[InternalPos.Index[0]] := 	RefPosHum[InternalPos.Index[0]]; // Due to a optical sensor fail reset the actual value of position to the referent position

		// Check if the Reflex sensors doesn't block the ball (if does, the sensing of position is not required _ just a momentary status)
		ELSIF (ExternalModulOK[InternalPos.Index[0]] = FALSE) THEN
					ActPosHumAxis[InternalPos.Index[0]] := 	InternalPos.CurrentPosition[InternalPos.Index[0]]; // Due to a reflex sensor fail reset the actual value of position to the referent position

			// Actual human position is set as a last
		ELSE
			ActPosHumAxis[InternalPos.Index[0]] := InternalPos.CurrentPosition[InternalPos.Index[0]]; // Last detected value in all other cases
		END_IF

	(*// Compute the positions all figures of opponent (by calling the function: DetPos_Figure)
	FOR InternalPos.Index[2] := 0 TO 3 DO

		// Set the input values into the function block
		InternalPos.DetPos_Figure0.ActPosHumAxisDP[InternalPos.Index[2]] := ActPosHumAxis[InternalPos.Index[2]];

		// Call the function block
		InternalPos.DetPos_Figure0();
	END_FOR;

	FOR InternalPos.Index[3] := 0 TO 10 DO

		// Call the output values of position all figures
		InternalPos.DetPos_Figure0.ActPosHumFigDP[InternalPos.Index[3]] := ActPosHumFig[InternalPos.Index[3]]*)
	END_FOR;

END_FUNCTION_BLOCK

		(* NUMERIC CALCULATION OF POSITION ALL AXES *)
FUNCTION_BLOCK DetPos_Figure

	// Set the value at position of Goalman Axis by the Actual Position of Axis with Displacement of Axis
	IF ActPosHumAxisDP[0] < MaxPosHumDP[0] AND ActPosHumAxisDP[0] > MinPosHumDP[0] THEN
		ActPosHumFigDP[0] := ActPosHumAxisDP[0]+DispAxisDP[0];
	ELSIF ActPosHumAxisDP[0] > MaxPosHumDP[0] THEN
		ActPosHumFigDP[0] := MaxPosHumDP[0];
	ELSIF ActPosHumAxisDP[0] < MinPosHumDP[0] THEN
		ActPosHumFigDP[0] := MinPosHumDP[0];
	ELSE
		ActPosHumFigDP[0] := ActPosHumAxisDP[0] + DispAxisDP[0];
	END_IF

	FOR i1 := 1 TO 2 DO
		// Set the value at position of Defender Axis by the Actual Position of Axis with Displacement of Axis
		IF ActPosHumAxisDP[1] < MaxPosHumDP[1] AND ActPosHumAxisDP[1] > MinPosHumDP[1] THEN
			ActPosHumFigDP[i1] := ActPosHumAxisDP[1]+ DispAxisDP[i1];
		ELSIF ActPosHumAxisDP[1] > MaxPosHumDP[1] THEN
			ActPosHumFigDP[i1] := MaxPosHumDP[1] + DispAxisDP[i1];
		ELSIF ActPosHumAxisDP[1] < MinPosHumDP[1] THEN
			ActPosHumFigDP[i1] := MinPosHumDP[1] + DispAxisDP[i1];
		ELSE
			ActPosHumFigDP[i1] := ActPosHumAxisDP[1] + DispAxisDP[i1];
		END_IF

	END_FOR;

	FOR i2 := 3 TO 7 DO
		// Set the value at position of Middle Defender Axis by the Actual Position of Axis with Displacement of Axis
		IF ActPosHumAxisDP[2] < MaxPosHumDP[2] AND ActPosHumAxisDP[2] > MinPosHumDP[2] THEN
			ActPosHumFigDP[i2] := ActPosHumAxisDP[2]+ DispAxisDP[i2];
		ELSIF ActPosHumAxisDP[2] > MaxPosHumDP[2] THEN
			ActPosHumFigDP[i2] := MaxPosHumDP[2] + DispAxisDP[i2];
		ELSIF ActPosHumAxisDP[2] < MinPosHumDP[2] THEN
			ActPosHumFigDP[i2] := MinPosHumDP[2] + DispAxisDP[i2];
		ELSE
			ActPosHumFigDP[i2] := ActPosHumAxisDP[2] + DispAxisDP[i2];
		END_IF

	END_FOR;

	FOR i3 := 8 TO 10 DO
		// Set the value at position of Forward Axis by the Actual Position of Axis with Displacement of Axis
		IF ActPosHumAxisDP[3] < MaxPosHumDP[3] AND ActPosHumAxisDP[3] > MinPosHumDP[3] THEN
			ActPosHumFigDP[i3] := ActPosHumAxisDP[3]+ DispAxisDP[i3];
		ELSIF ActPosHumAxisDP[3] > MaxPosHumDP[3] THEN
			ActPosHumFigDP[i3] := MaxPosHumDP[3] + DispAxisDP[i3];
		ELSIF ActPosHumAxisDP[3] < MinPosHumDP[3] THEN
			ActPosHumFigDP[i3] := MinPosHumDP[3] + DispAxisDP[i3];
		ELSE
			ActPosHumFigDP[i3] := ActPosHumAxisDP[3] + DispAxisDP[i3];
		END_IF

	END_FOR;

END_FUNCTION_BLOCK
```

### Types.typ - not listed in the package file held
```iecst
TYPE
	PositionStatus :
		(
		PosCalcPos, (*1*)
		PosInitial
		);
	Stuct_OptSensInternal : 	STRUCT
		TransConstant : ARRAY[0..3]OF INT;
		MaxPosHum : ARRAY[0..3]OF INT := [1025,1850,665,975];
		MinPosHum : ARRAY[0..3]OF INT := [-1025,-1850,-665,-975];
		RefPosHum : ARRAY[0..3]OF INT := [4(0)];
		MaxPosSens : ARRAY[0..3]OF INT := [26357,31402,29161,30516];
		MinPosSens : ARRAY[0..3]OF INT := [10382,6652,23050,12288];
		RefPosSens : ARRAY[0..3]OF INT := [19501,19027,26106,21401];
		Index : ARRAY[0..4]OF USINT;
		DR_ReflexSensStatus_0 : DetectionRotation;
		DP_Figure_0 : DetPos_Figure;
		MinAccDiff : INT := 100;
		MaxAccDiff : ARRAY[0..3]OF INT := [4(100)];
		CurrentPosition : ARRAY[0..3]OF INT;
	END_STRUCT;
	Stuct_RexlSensInternal : 	STRUCT
		ActReflexSensStatusRS : ARRAY[0..3]OF BOOL;
		ErrorStatusRS : ARRAY[0..3]OF BOOL;
		ExternalReflexSensStatusRS : ARRAY[0..3]OF BOOL;
		ReflexSensStatusRS : ARRAY[0..3]OF BOOL;
		IndexR : ARRAY[0..1]OF USINT;
	END_STRUCT;
	Struct_OptSensFigInternal : 	STRUCT
		MaxPosHumDP : ARRAY[0..3]OF INT;
		MinPosHumDP : ARRAY[0..3]OF INT;
		DispAxisDP : ARRAY[0..10]OF INT := [0,-1200,1200,-2400,-1200,0,1200,2400,-2100,0,2100];
		CurrentPosition : ARRAY[0..10]OF INT;
		Index : ARRAY[0..2]OF USINT;
	END_STRUCT;
END_TYPE
```

### RO_Sensors.fun - not listed in the package file held
```iecst
FUNCTION_BLOCK DetectionPositionAxis
	VAR_INPUT
		ActPosSens : ARRAY[0..3] OF INT;
		ErrorOptSens : ARRAY[0..3] OF BOOL;
		ReflexSensStatus : ARRAY[0..3] OF BOOL;
	END_VAR
	VAR_OUTPUT
		ActPosHumFig : ARRAY[0..10] OF INT;
		ActPosHumAxis : ARRAY[0..3] OF INT;
		ExternalReflexSensStatus : ARRAY[0..3] OF BOOL;
	END_VAR
	VAR
		InternalPos : Stuct_OptSensInternal;
	END_VAR
END_FUNCTION_BLOCK

FUNCTION_BLOCK DetectionRotation
	VAR_INPUT
		ErrorReflSensRS : ARRAY[0..3] OF BOOL;
		ReflexSensStatusRS : ARRAY[0..3] OF BOOL;
	END_VAR
	VAR_OUTPUT
		ExternalReflexSensStatusRS : ARRAY[0..3] OF BOOL;
		ActReflRotRS : ARRAY[0..3] OF BOOL;
	END_VAR
	VAR
		InternalRot : Stuct_RexlSensInternal;
	END_VAR
END_FUNCTION_BLOCK

FUNCTION_BLOCK DetPos_Figure
	VAR_INPUT
		ActPosHumAxisDP : ARRAY[0..3] OF INT;
	END_VAR
	VAR_OUTPUT
		ActPosHumFigDP : ARRAY[0..10] OF INT;
	END_VAR
	VAR
		InternalPosFig : Struct_OptSensFigInternal;
	END_VAR
END_FUNCTION_BLOCK
```

### DetectionPositionAxis.st - not listed in the package file held
```iecst
(* NUMERIC CALCULATION OF POSITION ALL AXES *)
FUNCTION_BLOCK DetectionPositionAxis

		// Calculate a constants
		InternalPos.TransConstant[0] := (InternalPos.MaxPosSens[0]-InternalPos.MinPosSens[0])/(InternalPos.MaxPosHum[0]-InternalPos.MinPosHum[0]);
		InternalPos.TransConstant[1] := (InternalPos.MaxPosSens[1]-InternalPos.MinPosSens[1])/(InternalPos.MaxPosHum[1]-InternalPos.MinPosHum[1]);
		InternalPos.TransConstant[2] := (InternalPos.MaxPosSens[2]-InternalPos.MinPosSens[2])/(InternalPos.MaxPosHum[2]-InternalPos.MinPosHum[2]);
		InternalPos.TransConstant[3] := (InternalPos.MaxPosSens[3]-InternalPos.MinPosSens[3])/(InternalPos.MaxPosHum[3]-InternalPos.MinPosHum[3]);

	// Check the status of Reflex sensors if they work well (TRUE = figure block the balon; FALSE = figure open the way)
	FOR InternalPos.Index[1] := 0 TO 3 DO

		InternalPos.DR_ReflexSensStatus_0.ReflexSensStatusRS[InternalPos.Index[1]] := ReflexSensStatus[InternalPos.Index[1]];
	END_FOR;

	// Calling FB DetRot_ModulOK_0
	InternalPos.DR_ReflexSensStatus_0();

	// Calculation state compute an atual value of distance or set the max/min value
	FOR InternalPos.Index[0] := 0 TO 3 DO

		// Set the External ModulOK value for case disfunction of
		ExternalReflexSensStatus[InternalPos.Index[0]] := InternalPos.DR_ReflexSensStatus_0.ExternalReflexSensStatusRS[InternalPos.Index[0]];

		// Optical sensor work well and values are in range and diference is over the minimal limit (compute a position by equation)
		IF (ErrorOptSens[InternalPos.Index[0]] = FALSE) AND ((ActPosSens[InternalPos.Index[0]] < InternalPos.MaxPosSens[InternalPos.Index[0]]) AND (ABS(ActPosSens[InternalPos.Index[0]] - InternalPos.CurrentPosition[InternalPos.Index[0]]) > InternalPos.MaxAccDiff[0])) AND ((ActPosSens[InternalPos.Index[0]] > InternalPos.MinPosSens[InternalPos.Index[0]]) AND (ABS(ActPosSens[InternalPos.Index[0]] - InternalPos.CurrentPosition[InternalPos.Index[0]]) > InternalPos.MaxAccDiff[0])) THEN
			ActPosHumAxis[InternalPos.Index[0]] := InternalPos.RefPosHum[InternalPos.Index[0]] + ((ActPosSens[InternalPos.Index[0]] - InternalPos.RefPosSens[InternalPos.Index[0]]) / InternalPos.TransConstant[InternalPos.Index[0]]);
			InternalPos.CurrentPosition[InternalPos.Index[0]] := ActPosHumAxis[InternalPos.Index[0]]; // Last detected value is safed as previous value for case Error mode of sensor

		// Optical sensor work well and values are in range and diference is in the minimal limit (set the previous value of position)
		ELSIF (ErrorOptSens[InternalPos.Index[0]] = FALSE) AND ((ActPosSens[InternalPos.Index[0]] < InternalPos.MaxPosSens[InternalPos.Index[0]]) AND (ABS(ActPosSens[InternalPos.Index[0]] - InternalPos.CurrentPosition[InternalPos.Index[0]]) < InternalPos.MaxAccDiff[0])) AND ((ActPosSens[InternalPos.Index[0]] > InternalPos.MinPosSens[InternalPos.Index[0]]) AND (ABS(ActPosSens[InternalPos.Index[0]] - InternalPos.CurrentPosition[InternalPos.Index[0]]) < InternalPos.MaxAccDiff[0])) THEN
			ActPosHumAxis[InternalPos.Index[0]]	:= InternalPos.CurrentPosition[InternalPos.Index[0]]; // Previous value of position

		// Optical sensor doesn't work well but values are in range
		ELSIF (ErrorOptSens[InternalPos.Index[0]] = TRUE) AND (ActPosSens[InternalPos.Index[0]] < InternalPos.MaxPosSens[InternalPos.Index[0]]) AND (ActPosSens[InternalPos.Index[0]] > InternalPos.MinPosSens[InternalPos.Index[0]]) THEN
			ActPosHumAxis[InternalPos.Index[0]] := 	InternalPos.CurrentPosition[InternalPos.Index[0]]; // Previous value of position

		// Optical sensor doesn't work well but values are over the maximum range
		ELSIF (ErrorOptSens[InternalPos.Index[0]] = TRUE) AND ((ActPosSens[InternalPos.Index[0]] > 500) OR (ActPosSens[InternalPos.Index[0]] < 8000))THEN
			ActPosHumAxis[InternalPos.Index[0]] := 	InternalPos.CurrentPosition[InternalPos.Index[0]]; // Previous value of position

		// Check if the Optical sensors are switched on (if not, sensored values are in range <-100 ; +100> _ the minimum limit sets InternalPos.MinAccDiff)
		ELSIF (ActPosSens[InternalPos.Index[0]] < InternalPos.MinAccDiff) THEN
			ActPosHumAxis[InternalPos.Index[0]] := 	InternalPos.RefPosHum[InternalPos.Index[0]]; // Due to a optical sensor fail set referent value of position by previous value of position

		// Check if the Reflex sensors doesn't block the ball (if does, the sensing of position is not required _ just a momentary status)
		ELSIF (ExternalReflexSensStatus[InternalPos.Index[0]] = FALSE) THEN
					ActPosHumAxis[InternalPos.Index[0]] := 	InternalPos.CurrentPosition[InternalPos.Index[0]]; // Due to a reflex sensor fail reset the actual value of position to the referent position

			// Actual human position is set as a last
		ELSE
			ActPosHumAxis[InternalPos.Index[0]] := InternalPos.RefPosHum[InternalPos.Index[0]]; // Set referent position in all other cases as default
		END_IF

	END_FOR;

	// Compute the positions all figures of opponent (by calling the function: DetPos_Figure)
	FOR InternalPos.Index[2] := 0 TO 3 DO

		// Set the input values into the function block
		InternalPos.DP_Figure_0.ActPosHumAxisDP[InternalPos.Index[2]] := ActPosHumAxis[InternalPos.Index[2]];

	END_FOR;

	// Call the function block
	InternalPos.DP_Figure_0();
	FOR InternalPos.Index[3] := 0 TO 10 DO

		// Call the output values of position all figures
 		ActPosHumFig[InternalPos.Index[3]] := InternalPos.DP_Figure_0.ActPosHumFigDP[InternalPos.Index[3]];

	END_FOR;

END_FUNCTION_BLOCK

		(* NUMERIC CALCULATION OF POSITION ALL AXES *)
FUNCTION_BLOCK DetPos_Figure

	// Set the value at position of Goalman Axis by the Actual Position of Axis with Displacement of Axis
	IF (ActPosHumAxisDP[0] < InternalPosFig.MaxPosHumDP[0]) AND (ActPosHumAxisDP[0] > InternalPosFig.MinPosHumDP[0]) THEN
		ActPosHumFigDP[0] := ActPosHumAxisDP[0] + InternalPosFig.DispAxisDP[0];
		InternalPosFig.CurrentPosition[0] := ActPosHumFigDP[0];
	//
	ELSIF ActPosHumAxisDP[0] > InternalPosFig.MaxPosHumDP[0] THEN
		ActPosHumFigDP[0] := InternalPosFig.MaxPosHumDP[0];

	//
	ELSIF ActPosHumAxisDP[0] < InternalPosFig.MinPosHumDP[0] THEN
		ActPosHumFigDP[0] := InternalPosFig.MinPosHumDP[0];

	//
	ELSE
		ActPosHumFigDP[0] := ActPosHumAxisDP[0] + InternalPosFig.DispAxisDP[0];
	END_IF

	FOR InternalPosFig.Index[0] := 1 TO 2 DO
		// Set the value at position of Defender Axis by the Actual Position of Axis with Displacement of Axis
		IF (ActPosHumAxisDP[1] < InternalPosFig.MaxPosHumDP[1]) AND (ActPosHumAxisDP[1] > InternalPosFig.MinPosHumDP[1]) THEN
			ActPosHumFigDP[InternalPosFig.Index[0]] := ActPosHumAxisDP[1] + InternalPosFig.DispAxisDP[InternalPosFig.Index[0]];
			InternalPosFig.CurrentPosition[InternalPosFig.Index[0]] := ActPosHumFigDP[InternalPosFig.Index[0]];
		//
		ELSIF ActPosHumAxisDP[1] > InternalPosFig.MaxPosHumDP[1] THEN
			ActPosHumFigDP[InternalPosFig.Index[0]] := InternalPosFig.MaxPosHumDP[1] + InternalPosFig.DispAxisDP[InternalPosFig.Index[0]];

		//
		ELSIF ActPosHumAxisDP[1] < InternalPosFig.MinPosHumDP[1] THEN
			ActPosHumFigDP[InternalPosFig.Index[0]] := InternalPosFig.MinPosHumDP[1] + InternalPosFig.DispAxisDP[InternalPosFig.Index[0]];

		//
		ELSE
			ActPosHumFigDP[InternalPosFig.Index[0]] := 	InternalPosFig.CurrentPosition[InternalPosFig.Index[0]];
		END_IF

	END_FOR;

	FOR InternalPosFig.Index[1] := 3 TO 7 DO
		// Set the value at position of Middle Defender Axis by the Actual Position of Axis with Displacement of Axis
		IF (ActPosHumAxisDP[2] < InternalPosFig.MaxPosHumDP[2]) AND (ActPosHumAxisDP[2] > InternalPosFig.MinPosHumDP[2]) THEN
			ActPosHumFigDP[InternalPosFig.Index[1]] := ActPosHumAxisDP[2] + InternalPosFig.DispAxisDP[InternalPosFig.Index[1]];
			InternalPosFig.CurrentPosition[InternalPosFig.Index[1]] := ActPosHumFigDP[InternalPosFig.Index[1]];
		//
		ELSIF ActPosHumAxisDP[2] > InternalPosFig.MaxPosHumDP[2] THEN
			ActPosHumFigDP[InternalPosFig.Index[1]] := InternalPosFig.MaxPosHumDP[2] + InternalPosFig.DispAxisDP[InternalPosFig.Index[1]];

		//
		ELSIF ActPosHumAxisDP[2] < InternalPosFig.MinPosHumDP[2] THEN
			ActPosHumFigDP[InternalPosFig.Index[1]] := InternalPosFig.MinPosHumDP[2] + InternalPosFig.DispAxisDP[InternalPosFig.Index[1]];

		//
		ELSE
			ActPosHumFigDP[InternalPosFig.Index[1]] := InternalPosFig.CurrentPosition[InternalPosFig.Index[1]];
		END_IF

	END_FOR;

	FOR InternalPosFig.Index[2] := 8 TO 10 DO
		// Set the value at position of Forward Axis by the Actual Position of Axis with Displacement of Axis
		IF (ActPosHumAxisDP[3] < InternalPosFig.MaxPosHumDP[3]) AND (ActPosHumAxisDP[3] > InternalPosFig.MinPosHumDP[3]) THEN
			ActPosHumFigDP[InternalPosFig.Index[2]] := ActPosHumAxisDP[3]+ InternalPosFig.DispAxisDP[InternalPosFig.Index[2]];
			InternalPosFig.CurrentPosition[InternalPosFig.Index[2]] := ActPosHumFigDP[InternalPosFig.Index[2]];
		//
		ELSIF ActPosHumAxisDP[3] > InternalPosFig.MaxPosHumDP[3] THEN
			ActPosHumFigDP[InternalPosFig.Index[2]] := InternalPosFig.MaxPosHumDP[3] + InternalPosFig.DispAxisDP[InternalPosFig.Index[2]];

		//
		ELSIF ActPosHumAxisDP[3] < InternalPosFig.MinPosHumDP[3] THEN
			ActPosHumFigDP[InternalPosFig.Index[2]] := InternalPosFig.MinPosHumDP[3] + InternalPosFig.DispAxisDP[InternalPosFig.Index[2]];

		//
		ELSE
			ActPosHumFigDP[InternalPosFig.Index[2]] := InternalPosFig.CurrentPosition[InternalPosFig.Index[2]];
		END_IF

	END_FOR;

END_FUNCTION_BLOCK
```

### Library Logical/Libraries/RO_Sensors/ro_sensors (IEC)
